// TIA Portal project "XSFW_TIA31001_B0_V15.1" (V15.1)

(* hardware
DEVICE "S7-1200 station_1"  S7-1200 Station
   slot 0: "Rack_0"  S7-1200 Rack  Rack  V1.0
   slot 1: "PLC_Divider"  CPU 1214C DC/DC/DC  6ES7 214-1AG40-0XB0  V4.2
   slot 2: "DI 16/DQ 16x24VDC_1"  6ES7 223-1BL32-0XB0  V2.0
   slot 3: "AI 4x13BIT/AQ 2x14BIT_1"  6ES7 234-4HE32-0XB0  V2.0
   slot 101: "CM 1242-5"  CM 1242-5  6GK7 242-5DX30-0XE0  V1.0
DEVICE "CSM"  SCALANCE X-Station
   slot 0: "Bastidor SCALANCE X"  Rail
   slot 0: "Switch"  6GK7 277-1AA00-0AA0
DEVICE "HMI_1"  KTP700 Basic PN
   slot 0: "HMI_1"  KTP700 Basic PN  6AV2 123-2GB03-0AX0  15.0.0.0
   slot 1: "HMI_RT_1"  KTP700 Basic PN  6AV2 123-2GB03-0AX0  15.0.0.0
   slot 5: "HMI_1.IE_CP_1"  PROFINET Interface  15.0.0.0
      slot 1: "Interfaz PROFINET_1"  PROFINET Interface
         slot 1: "Port_1"  Port
DEVICE "Dispositivo GSD_1"  GSD.Device.PN
   slot 0: "Rack"  Rack  V1.0
   slot 0: "V90-X"  SINAMICS V90 PN V1.0  6SL3 210-5Fxxx-xxFx  V1.00
      slot 0: "SINAMICS V90 PN V1.0"  SINAMICS V90 PN V1.0
      slot 1: "PN-IO"  PN-IO
         slot 1: "Puerto 1"  Port 1
         slot 2: "Puerto 2"  Port 2
      slot 1: "Drive"  Drive
         slot 0: "Punto de acceso a módulo"  Module Access Point
         slot 1: "sin PROFIsafe"  without PROFIsafe
   slot 2: "Telegrama estándar 3, PZD-5/9"  Standard telegram 3, PZD-5/9
DEVICE "Dispositivo GSD_2"  GSD.Device.PN
   slot 0: "Rack"  Rack  V1.0
   slot 0: "V90-Y"  SINAMICS V90 PN V1.0  6SL3 210-5Fxxx-xxFx  V1.00
      slot 0: "SINAMICS V90 PN V1.0"  SINAMICS V90 PN V1.0
      slot 1: "PN-IO"  PN-IO
         slot 1: "Puerto 1"  Port 1
         slot 2: "Puerto 2"  Port 2
      slot 1: "Drive"  Drive
         slot 0: "Punto de acceso a módulo"  Module Access Point
         slot 1: "sin PROFIsafe"  without PROFIsafe
   slot 2: "Telegrama estándar 3, PZD-5/9"  Standard telegram 3, PZD-5/9
*)

// ===== PLC "PLC_Divider"  CPU 1214C DC/DC/DC =====

VAR_GLOBAL   // PLC tag table "Tabla de variables estándar"
   "iCntBot" AT %I0.3 : Bool;
   "iSnsBotBaj" AT %I0.4 : Bool;
   "iSnsBotAlt" AT %I0.5 : Bool;
   "iCH_A" AT %I0.0 : Bool;
   "iCH_B" AT %I0.1 : Bool;
   "iCH_Z" AT %I0.2 : Bool;
   "iSns_Ch1Full" AT %I0.6 : Bool;
   "iSns_Ch2Full" AT %I3.6 : Bool;
   "iSns_Ch3Full" AT %I3.7 : Bool;
   "iSign_HabInv" AT %I3.0 : Bool;
   "iPul_Marcha" AT %I3.1 : Bool;
   "iPul_Parada" AT %I3.2 : Bool;
   "iPul_Rst" AT %I3.3 : Bool;
   "iProt_Abiertas" AT %I3.4 : Bool;
   "iTrip_Inverter" AT %I3.5 : Bool;
   "iRef_Analog" AT %IW54 : Int;
   "qRev_Alarma" AT %Q0.0 : Bool;
   "qSem_Verde" AT %Q0.1 : Bool;
   "qSem_rojo" AT %Q0.2 : Bool;
   "qTest_Marcha" AT %Q0.3 : Bool;
   "qRes_Alarma" AT %Q0.4 : Bool;
   "qRes_Inversor" AT %Q0.5 : Bool;
   "qFwd_Inversor" AT %Q0.6 : Bool;
   "qTrig_2" AT %Q0.7 : Bool;
   "qSign_Marcha" AT %Q1.0 : Bool;
   "qSign_Falla" AT %Q1.1 : Bool;
   "qTrig_1" AT %Q2.0 : Bool;
   "qTrig_22" AT %Q2.1 : Bool;
   "qRef_Analog" AT %IW82 : Int;
   "System_Byte" AT %MB1 : Byte;
   "FirstScan" AT %M1.0 : Bool;
   "DiagStatusUpdate" AT %M1.1 : Bool;
   "AlwaysTRUE" AT %M1.2 : Bool;
   "AlwaysFALSE" AT %M1.3 : Bool;
   "Clock_Byte" AT %MB0 : Byte;
   "Clock_10Hz" AT %M0.0 : Bool;
   "Clock_5Hz" AT %M0.1 : Bool;
   "Clock_2.5Hz" AT %M0.2 : Bool;
   "Clock_2Hz" AT %M0.3 : Bool;
   "Clock_1.25Hz" AT %M0.4 : Bool;
   "Clock_1Hz" AT %M0.5 : Bool;
   "Clock_0.625Hz" AT %M0.6 : Bool;
   "Clock_0.5Hz" AT %M0.7 : Bool;
   "Eje_Y_Drive_OUT" AT %Q74.0 : "PD_TEL3_OUT";
   "Eje_1_Drive_IN" AT %I68.0 : "PD_TEL3_IN";
   "Eje_1_Drive_OUT" AT %Q64.0 : "PD_TEL3_OUT";
   "MMovX" AT %M850.0 : Bool;
   "MMovXN" AT %M850.1 : Bool;
   "MMov2X" AT %M850.2 : Bool;
   "MMov2XN" AT %M850.3 : Bool;
   "MMovY" AT %M850.4 : Bool;
   "MMovYN" AT %M850.5 : Bool;
   "Eje_Y_Drive_IN(1)" AT %I86.0 : "PD_TEL3_IN";
   "Marca_Reset" AT %M103.0 : Bool;
   "SR_AlarmaOn" AT %M103.1 : Bool;
   "iHsc_Z" AT %ID1000 : DInt;
   "Hsc_Za" AT %MD20 : DInt;
   "Contando" AT %M150.0 : Bool;
   "Halt_Motor" AT %M150.2 : Bool;
   "Band_E24" AT %M150.3 : Bool;
   "Band_E22" AT %M150.4 : Bool;
   "Band_E23" AT %M150.5 : Bool;
   "Hsc_Zb" AT %MD28 : DInt;
   "Hsc_sub" AT %MD32 : DInt;
   "Hsc_sub1" AT %MD36 : DInt;
   "Enc_hab" AT %E104.0 : Bool;
   "Enc_stop" AT %I104.1 : Bool;
   "iEnc_Word1" AT %IW104 : Word;
   "iEnc_Word2" AT %IW106 : Word;
   "iEnc_Word3" AT %IW108 : Word;
   "iEnc_Word4" AT %IW110 : Word;
   "qEnc_Word5" AT %QW104 : Word;
   "qEnc_Word6" AT %QW106 : Word;
   "qEnc_Word7" AT %QW108 : Word;
   "qEnc_Word8" AT %QW110 : Word;
   "iSns_FinCarrX1" AT %I2.0 : Bool;
   "iSns_FinCarrX2" AT %I2.1 : Bool;
   "iSns_FinCarrY1" AT %I2.2 : Bool;
   "iSns_FinCarrY2" AT %I2.3 : Bool;
END_VAR

VAR_GLOBAL   // PLC tag table "Alarmas"
   "Alarmas_1" AT %MW100 : Word;
   "ProteccionAbierta" AT %M100.0 : Bool;
   "BotellaCaida" AT %M100.1 : Bool;
   "Fin_Carrera_X" AT %M100.4 : Bool;
   "Fin_Carrera_Y" AT %M100.5 : Bool;
   "Trip_Inverter" AT %M100.2 : Bool;
   "Error_Velocidad" AT %M100.3 : Bool;
END_VAR

VAR_GLOBAL   // PLC tag table "Inicializaciòn"
   "Marcas para la inicializaciòn" AT %MW102 : Word;
   "Start" AT %M102.0 : Bool;
END_VAR

DATA_BLOCK "01_LINEA_Entradas-DB"   // DB1
{ S7_Optimized_Access := 'TRUE' }
VERSION : 0.1
   VAR
      Contador : Bool;   // Pulsador de marcha
      Sensor_Bajo : Bool;   // Pulsador de parada
      Sensor_Alto : Bool;   // Pulsador de marcha columna 4
      CH_A : Bool;   // Pulsador de parada de emergancia columna 4
      CH_B : Bool;   // Pulsador de marcha columna 6
      CH_Z : Bool;   // Pulsador de parada de emergancia columna 6
      Canal1_Full : Bool;   // Pulsador de marcha columna 9
      Canal2_Full : Bool;   // Pulsador de parada de emergancia columna 9
      Canal3_Full : Bool;   // Pulsador de marcha columna 11
      Hab_Inverter : Bool;   // Pulsador de parada de emergancia columna 11
      Marcha : Bool;   // Pulsador de marcha columna 12
      Parada : Bool;   // Pulsador de parada de emergancia columna 12
      Reset : Bool;   // Pulsador de parada de emergancia del tablero general
      Protecciones_Abiertas : Bool;   // Pulsador de parada de emergencia del tablero de la fosa
      Trip_Inverter : Bool;   // Señal de falla del variador
      Enc_andando : Bool;
      Enc_parada : Bool;
   END_VAR
BEGIN
END_DATA_BLOCK

DATA_BLOCK "02_LINEA_Salidas-DB"   // DB2
{ S7_Optimized_Access := 'TRUE' }
VERSION : 0.1
   VAR
      Alarma_Sonora : Bool;   // Marcha para el variador
      Semaforo_Verde : Bool;   // Sentido adelante variador
      Semaforo_Rojo : Bool;   // Sentido atras variador
      Testigo_Marcha : Bool;   // Indicador sonoro
      Reset_Alarma : Bool;   // Indicador de linea en marcha
      Reset_Inverter : Bool;   // Indicador de linea parada
      Avance_Inverter : Bool;   // Buzzer de la baliza del tablero principal
      Trigger_2 : Bool;   // Lampara verde de la baliza del tablero principal
      EnMarcha : Bool;   // Lampara roja de la baliza del tablero principal
      EnFalla : Bool;   // Lampara amarilla de la baliza del tablero principal
      Trigger_11 : Bool;
      Trigger_22 : Bool;
      Ref_20mA : Int;
   END_VAR
BEGIN
END_DATA_BLOCK

DATA_BLOCK "MotorInverter"   // DB5
{ S7_Optimized_Access := 'TRUE' }
VERSION : 0.1
// stored: InstanceOfName Motor Simple
"Motor Simple"
BEGIN
END_DATA_BLOCK

DATA_BLOCK "FB_INC_GENERAL_DB"   // DB7
{ S7_Optimized_Access := 'FALSE' }
VERSION : 0.1
// stored: InstanceOfName FB_INC_GENERAL
"FB_INC_GENERAL"
BEGIN
END_DATA_BLOCK

DATA_BLOCK "Cuentas_Matematicas1_DB"   // DB15
{ S7_Optimized_Access := 'TRUE' }
VERSION : 0.1
   VAR
      MovXNeg : Real := 0.0;
      Mov2X : Real := 0.0;
      Mov2XNeg : Real := 0.0;
      MovYNeg : Real := 0.0;
   END_VAR
BEGIN
END_DATA_BLOCK

DATA_BLOCK "FB_GENERAL_DB"   // DB17
{ S7_Optimized_Access := 'FALSE' }
VERSION : 0.1
// stored: InstanceOfName FB_SUB_1_GENERAL
"FB_SUB_1_GENERAL"
BEGIN
END_DATA_BLOCK

DATA_BLOCK "Cuentas_Matematicas1_DB_1"   // DB20
{ S7_Optimized_Access := 'TRUE' }
VERSION : 0.1
// stored: InstanceOfName Cuentas_Matematicas1
"Cuentas_Matematicas1"
BEGIN
END_DATA_BLOCK

DATA_BLOCK "DB_Encajonadora"   // DB28
{ S7_Optimized_Access := 'TRUE' }
VERSION : 0.1
   VAR
      Word1 : Word;   // bit 0 y 1 para guardar estado de encajonadora
      Word2 : Word;
      Word3 : Word;
      Word4 : Word;
      Word5 : Word;
      Word6 : Word;
      Word7 : Word;
      Word8 : Word;
   END_VAR
BEGIN
END_DATA_BLOCK

DATA_BLOCK "FB_SUB_1_GENERAL_DB"   // DB35
{ S7_Optimized_Access := 'FALSE' }
VERSION : 0.1
// stored: InstanceOfName FB_SUB_1_GENERAL
"FB_SUB_1_GENERAL"
BEGIN
END_DATA_BLOCK

DATA_BLOCK "FB_SUB_0_GENERAL_DB"   // DB36
{ S7_Optimized_Access := 'TRUE' }
VERSION : 0.1
// stored: InstanceOfName FB_SUB_0_GENERAL
"FB_SUB_0_GENERAL"
BEGIN
END_DATA_BLOCK

DATA_BLOCK "DB_SUB_1_GENERAL"   // DB100
{ S7_Optimized_Access := 'FALSE' }
VERSION : 0.1
// stored: InstanceOfName FB_SUB_1_GENERAL
"FB_SUB_1_GENERAL"
BEGIN
END_DATA_BLOCK

// folder: COMANDOS

DATA_BLOCK "DB_SUB_0_COM_GENERAL"   // DB600
{ S7_Optimized_Access := 'FALSE' }
VERSION : 0.1
   VAR
      ManipEsperaCarro : Bool;
      RecepCarroConfir : Bool;
      SalidaEsperaCarro1 : Bool;
      SalidaEsperaCarro2 : Bool;
      TengoCarroEnPortacarro : Bool;
      ReconocimientoAlarmas : Bool;
   END_VAR
BEGIN
END_DATA_BLOCK

// folder: INCIDENTES

DATA_BLOCK "DB_INC_GENERAL"   // DB500
{ S7_Optimized_Access := 'FALSE' }
VERSION : 0.1
// stored: InstanceOfName FB_INC_GENERAL
"FB_INC_GENERAL"
BEGIN
END_DATA_BLOCK

// folder: PUESTA EN MARCHA

DATA_BLOCK "DB_PUESTA_MARCHA"   // DB10
{ S7_Optimized_Access := 'TRUE' }
VERSION : 0.1
   VAR RETAIN
      MovYmm : Real := 30.0;
      MovXmm : Real := 30.0;
   END_VAR
   VAR
      TChFull : Time := T#1S;
   END_VAR
BEGIN
END_DATA_BLOCK

// folder: System blocks/Program resources

DATA_BLOCK "IEC_Counter_0_DB"   // DB6
{ S7_Optimized_Access := 'TRUE' }
AUTHOR : Simatic
FAMILY : IEC
NAME : CNTR
VERSION : 1.0
// stored: InstanceOfName IEC_COUNTER
"IEC_COUNTER"
BEGIN
END_DATA_BLOCK

DATA_BLOCK "IEC_Counter_1_DB"   // DB8
{ S7_Optimized_Access := 'TRUE' }
AUTHOR : Simatic
FAMILY : IEC
NAME : CNTR
VERSION : 1.0
// stored: InstanceOfName IEC_COUNTER
"IEC_COUNTER"
BEGIN
END_DATA_BLOCK

DATA_BLOCK "IEC_Counter_2_DB"   // DB9
{ S7_Optimized_Access := 'TRUE' }
AUTHOR : Simatic
FAMILY : IEC
NAME : CNTR
VERSION : 1.0
// stored: InstanceOfName IEC_COUNTER
"IEC_COUNTER"
BEGIN
END_DATA_BLOCK

DATA_BLOCK "IEC_Timer_ChFull"   // DB11
{ S7_Optimized_Access := 'TRUE' }
AUTHOR : Simatic
FAMILY : IEC
NAME : IEC_TMR
VERSION : 1.0
// stored: InstanceOfName IEC_TIMER
"IEC_TIMER"
BEGIN
END_DATA_BLOCK

DATA_BLOCK "IEC_Timer_0_DB_1"   // DB30
{ S7_Optimized_Access := 'TRUE' }
AUTHOR : Simatic
FAMILY : IEC
NAME : IEC_TMR
VERSION : 1.0
// stored: InstanceOfName IEC_TIMER
"IEC_TIMER"
BEGIN
END_DATA_BLOCK

DATA_BLOCK "IEC_Timer_0_DB_2"   // DB31
{ S7_Optimized_Access := 'TRUE' }
AUTHOR : Simatic
FAMILY : IEC
NAME : IEC_TMR
VERSION : 1.0
// stored: InstanceOfName IEC_TIMER
"IEC_TIMER"
BEGIN
END_DATA_BLOCK

DATA_BLOCK "IEC_Timer_0_DB_3"   // DB32
{ S7_Optimized_Access := 'TRUE' }
AUTHOR : Simatic
FAMILY : IEC
NAME : IEC_TMR
VERSION : 1.0
// stored: InstanceOfName IEC_TIMER
"IEC_TIMER"
BEGIN
END_DATA_BLOCK

DATA_BLOCK "IEC_Timer_0_DB_4"   // DB33
{ S7_Optimized_Access := 'TRUE' }
AUTHOR : Simatic
FAMILY : IEC
NAME : IEC_TMR
VERSION : 1.0
// stored: InstanceOfName IEC_TIMER
"IEC_TIMER"
BEGIN
END_DATA_BLOCK

DATA_BLOCK "IEC_Timer_0_DB_5"   // DB34
{ S7_Optimized_Access := 'TRUE' }
AUTHOR : Simatic
FAMILY : IEC
NAME : IEC_TMR
VERSION : 1.0
// stored: InstanceOfName IEC_TIMER
"IEC_TIMER"
BEGIN
END_DATA_BLOCK

// folder: VISUALIZACION

DATA_BLOCK "DB_VIS_GENERAL"   // DB800
{ S7_Optimized_Access := 'FALSE' }
VERSION : 0.1
   VAR
      CantBot : Int;
      AlarmaProtecciòn : Bool;
      AlarmaBotellaCaida : Bool;
      MC_Pwr_EnX : Bool;
      MC_Pwrt_EnY : Bool;
      MC_Res_ExX : Bool;
      MC_Res_ExY : Bool;
      MC_JogFwd_X : Bool;
      MC_JogFwd_Y : Bool;
      MC_JogBwd_X : Bool;
      MC_JogBwd_Y : Bool;
      HomingOk : Bool;
      Reset : Bool;
      Start : Bool;
   END_VAR
BEGIN
END_DATA_BLOCK

// folder: (top level)

DATA_BLOCK "Eje_Y"   // DB4, Motion_DB
{ S7_Optimized_Access := 'TRUE' }
AUTHOR : SIMATIC
FAMILY : BasicMC
NAME : TO_PosAx
VERSION : 6.0
// stored: InstanceOfName TO_PositioningAxis
"TO_PositioningAxis"
BEGIN
   // Axis.Encoder.TelegramAddressOutCU = %Q74.0
   // Axis.Encoder.TelegramAddressInCU = %I86.0
   // Axis.Encoder.DoNameCU = V90-Y.Drive_Encóder1
   // Axis.Drive.TelegramAddressOutCU = %Q74.0
   // Axis.Drive.TelegramAddressInCU = %I86.0
   // Axis.Drive.TelegramType = 2
   // Axis.Drive.DoNameCU = V90-Y.Drive
   // Axis.LengthUnitNormalized.Time = 1
   // Axis.LengthUnitNormalized.Distance = -2
   // Axis.Encoder.SelectedHscIndexCU = -1
   // Axis.Encoder.DbTypeCU = Classic
   // Axis.Drive.DbTypeCU = Classic
END_DATA_BLOCK

DATA_BLOCK "Eje_X"   // DB12, Motion_DB
{ S7_Optimized_Access := 'TRUE' }
AUTHOR : SIMATIC
FAMILY : BasicMC
NAME : TO_PosAx
VERSION : 6.0
// stored: InstanceOfName TO_PositioningAxis
"TO_PositioningAxis"
BEGIN
   // Axis.Encoder.TelegramAddressOutCU = %Q64.0
   // Axis.Encoder.TelegramAddressInCU = %I68.0
   // Axis.Encoder.DoNameCU = V90-X.Drive_Encóder1
   // Axis.Drive.TelegramAddressOutCU = %Q64.0
   // Axis.Drive.TelegramAddressInCU = %I68.0
   // Axis.Drive.TelegramType = 2
   // Axis.Drive.DoNameCU = V90-X.Drive
   // Axis.LengthUnitNormalized.Distance = 1013
   // Axis.Encoder.SelectedHscIndexCU = -1
   // Axis.Encoder.DbTypeCU = Classic
   // Axis.Drive.DbTypeCU = Classic
END_DATA_BLOCK

FUNCTION_BLOCK "Cuentas_Matematicas1"   // FB1, LAD
TITLE = ---------------------------Calculo de distancias----------------------------------------
{ S7_Optimized_Access := 'TRUE' }
VERSION : 0.1
BEGIN

REGION Network 1: Movimiento negativo en X
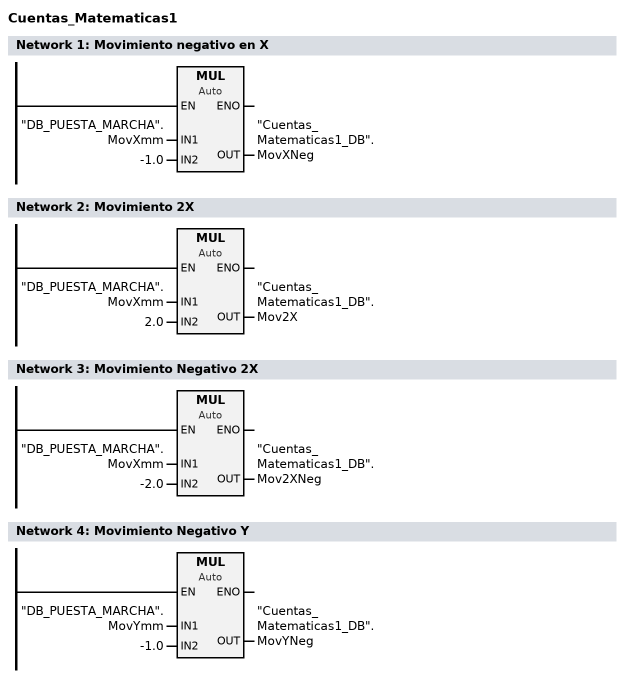
   RUNG wire#powerrail
      Mul(in1 := "DB_PUESTA_MARCHA".MovXmm, in2 := -1.0, out => "Cuentas_Matematicas1_DB".MovXNeg)
   END_RUNG
   // the same network as SCL:
   "Cuentas_Matematicas1_DB".MovXNeg := "DB_PUESTA_MARCHA".MovXmm * (-1.0);
END_REGION

REGION Network 2: Movimiento 2X
   RUNG wire#powerrail
      Mul(in1 := "DB_PUESTA_MARCHA".MovXmm, in2 := 2.0, out => "Cuentas_Matematicas1_DB".Mov2X)
   END_RUNG
   // the same network as SCL:
   "Cuentas_Matematicas1_DB".Mov2X := "DB_PUESTA_MARCHA".MovXmm * 2.0;
END_REGION

REGION Network 3: Movimiento Negativo 2X
   RUNG wire#powerrail
      Mul(in1 := "DB_PUESTA_MARCHA".MovXmm, in2 := -2.0, out => "Cuentas_Matematicas1_DB".Mov2XNeg)
   END_RUNG
   // the same network as SCL:
   "Cuentas_Matematicas1_DB".Mov2XNeg := "DB_PUESTA_MARCHA".MovXmm * (-2.0);
END_REGION

REGION Network 4: Movimiento Negativo Y
   RUNG wire#powerrail
      Mul(in1 := "DB_PUESTA_MARCHA".MovYmm, in2 := -1.0, out => "Cuentas_Matematicas1_DB".MovYNeg)
   END_RUNG
   // the same network as SCL:
   "Cuentas_Matematicas1_DB".MovYNeg := "DB_PUESTA_MARCHA".MovYmm * (-1.0);
END_REGION
END_FUNCTION_BLOCK

FUNCTION_BLOCK "FB_SUB_0_GENERAL"   // FB3, LAD
{ S7_Optimized_Access := 'TRUE' }
VERSION : 0.1
BEGIN

REGION Network 1
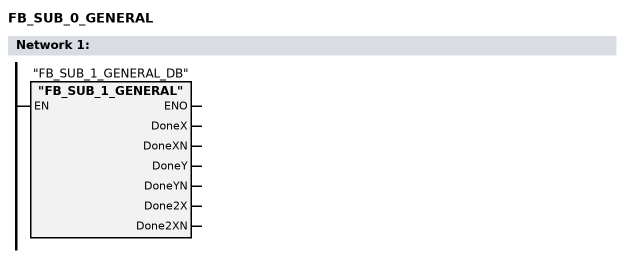
   RUNG wire#powerrail
      "FB_SUB_1_GENERAL_DB"(DoneX =>, DoneXN =>, DoneY =>, DoneYN =>, Done2X =>, Done2XN =>)
   END_RUNG
   // the same network as SCL:
   "FB_SUB_1_GENERAL_DB"();   // "FB_SUB_1_GENERAL"
END_REGION
END_FUNCTION_BLOCK

FUNCTION_BLOCK "FB_SUB_1_GENERAL"   // FB100, LAD
{ S7_Optimized_Access := 'FALSE' }
VERSION : 0.1
   VAR_OUTPUT
      DoneX : Bool;
      DoneXN : Bool;
      DoneY : Bool;
      DoneYN : Bool;
      Done2X : Bool;
      Done2XN : Bool;
   END_VAR
   VAR
      Estados : Array[0..32] of Bool;
      Concatenadoras : Array[0..32] of Bool;
      Prioritarias : Array[0..32] of Bool;
      Error_Concatenadoras : Bool;
      Error_Prioritarias : Bool;
      Cuenta_1 : Bool;
      Cuenta_2 : Bool;
      Cuenta_3 : Bool;
      "Cont_Botellas/2" : Int;
   END_VAR
BEGIN

REGION Network 1: Inicializaciòn
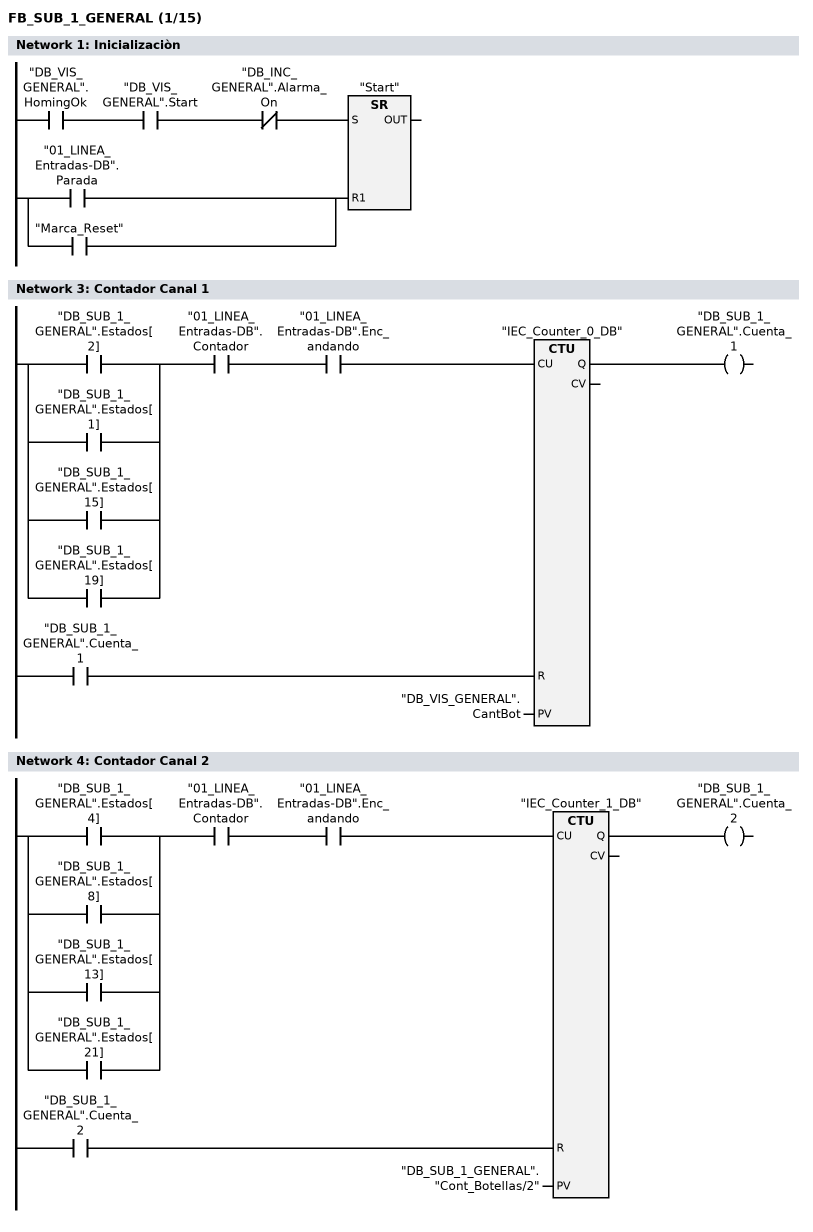
   RUNG wire#powerrail
      Contact( "DB_VIS_GENERAL".HomingOk )
      Contact( "DB_VIS_GENERAL".Start )
      I_Contact( "DB_INC_GENERAL".Alarma_On )
      S_SR(operand := "Start", r1 := wire#w1)
   END_RUNG
   RUNG wire#powerrail
      Contact( "01_LINEA_Entradas-DB".Parada )
   END_RUNG wire#w1
   RUNG wire#powerrail
      Contact( "Marca_Reset" )
   END_RUNG wire#w1
   // the same network as SCL:
   IF "DB_VIS_GENERAL".HomingOk AND "DB_VIS_GENERAL".Start AND NOT "DB_INC_GENERAL".Alarma_On THEN
       "Start" := TRUE;   // SR flip-flop
   END_IF;
   IF "01_LINEA_Entradas-DB".Parada OR "Marca_Reset" THEN "Start" := FALSE; END_IF;
END_REGION

REGION Network 2: -----------------OTROS---------------
END_REGION

REGION Network 3: Contador Canal 1
   "IEC_Counter_0_DB".CTU(CU := ("DB_SUB_1_GENERAL".Estados[2] OR "DB_SUB_1_GENERAL".Estados[1] OR "DB_SUB_1_GENERAL".Estados[15] OR "DB_SUB_1_GENERAL".Estados[19]) AND "01_LINEA_Entradas-DB".Contador AND "01_LINEA_Entradas-DB".Enc_andando,
                          R := "DB_SUB_1_GENERAL".Cuenta_1,
                          PV := "DB_VIS_GENERAL".CantBot);
   "DB_SUB_1_GENERAL".Cuenta_1 := "IEC_Counter_0_DB".Q;
END_REGION

REGION Network 4: Contador Canal 2
   "IEC_Counter_1_DB".CTU(CU := ("DB_SUB_1_GENERAL".Estados[4] OR "DB_SUB_1_GENERAL".Estados[8] OR "DB_SUB_1_GENERAL".Estados[13] OR "DB_SUB_1_GENERAL".Estados[21]) AND "01_LINEA_Entradas-DB".Contador AND "01_LINEA_Entradas-DB".Enc_andando,
                          R := "DB_SUB_1_GENERAL".Cuenta_2,
                          PV := "DB_SUB_1_GENERAL"."Cont_Botellas/2");
   "DB_SUB_1_GENERAL".Cuenta_2 := "IEC_Counter_1_DB".Q;
END_REGION

REGION Network 5: CASO I CANAL 2
   // Caso en el cual CH1/2 no estan llenos y hay que repartir solo la mitad de las botellas en canal central
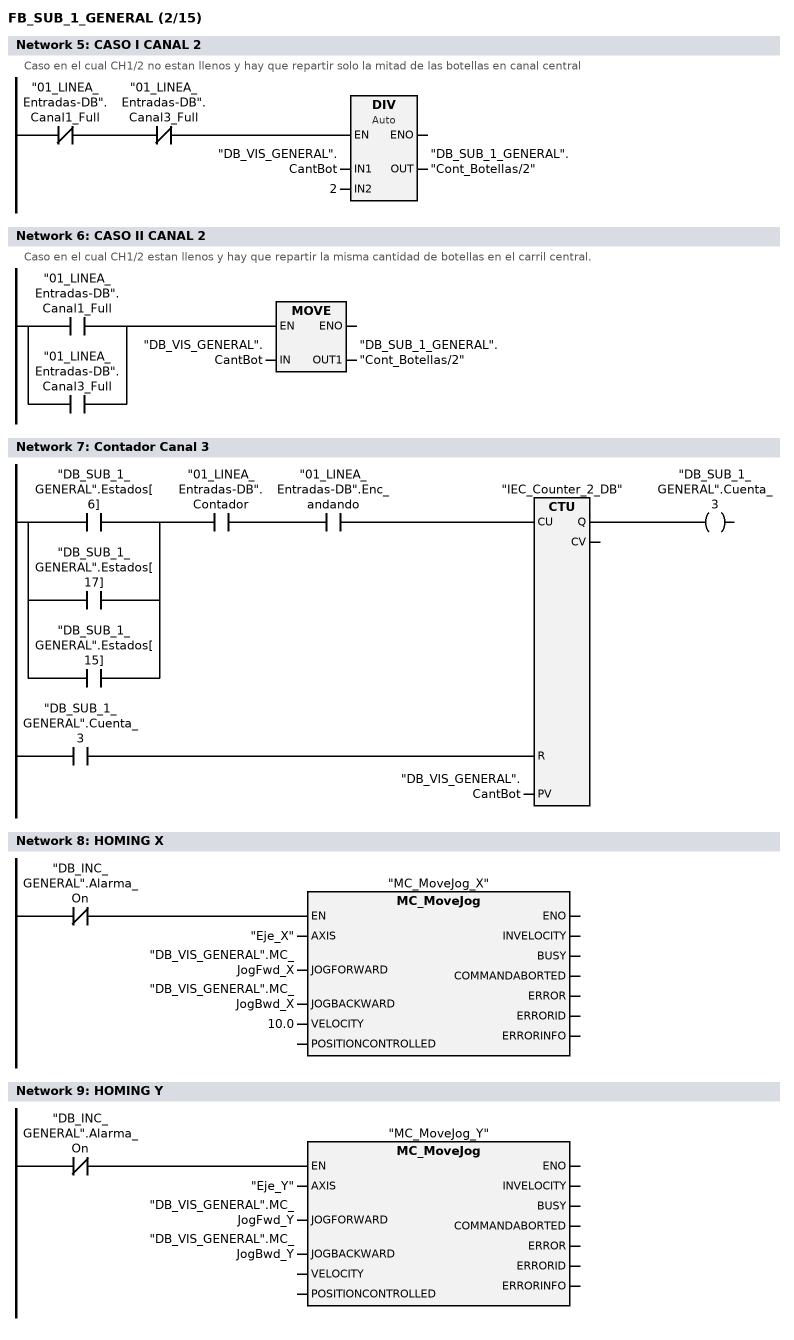
   RUNG wire#powerrail
      I_Contact( "01_LINEA_Entradas-DB".Canal1_Full )
      I_Contact( "01_LINEA_Entradas-DB".Canal3_Full )
      Div(in1 := "DB_VIS_GENERAL".CantBot, in2 := 2, out => "DB_SUB_1_GENERAL"."Cont_Botellas/2")
   END_RUNG
   // the same network as SCL:
   IF NOT "01_LINEA_Entradas-DB".Canal1_Full AND NOT "01_LINEA_Entradas-DB".Canal3_Full THEN
       "DB_SUB_1_GENERAL"."Cont_Botellas/2" := "DB_VIS_GENERAL".CantBot / 2;
   END_IF;
END_REGION

REGION Network 6: CASO II CANAL 2
   // Caso en el cual CH1/2 estan llenos y hay que repartir la misma cantidad de botellas en el carril central.
   RUNG wire#powerrail
      Contact( "01_LINEA_Entradas-DB".Canal1_Full )
      wire#w1
      Move(in := "DB_VIS_GENERAL".CantBot, out1 => "DB_SUB_1_GENERAL"."Cont_Botellas/2")
   END_RUNG
   RUNG wire#powerrail
      Contact( "01_LINEA_Entradas-DB".Canal3_Full )
   END_RUNG wire#w1
   // the same network as SCL:
   IF "01_LINEA_Entradas-DB".Canal1_Full OR "01_LINEA_Entradas-DB".Canal3_Full THEN
       "DB_SUB_1_GENERAL"."Cont_Botellas/2" := "DB_VIS_GENERAL".CantBot;
   END_IF;
END_REGION

REGION Network 7: Contador Canal 3
   "IEC_Counter_2_DB".CTU(CU := ("DB_SUB_1_GENERAL".Estados[6] OR "DB_SUB_1_GENERAL".Estados[17] OR "DB_SUB_1_GENERAL".Estados[15]) AND "01_LINEA_Entradas-DB".Contador AND "01_LINEA_Entradas-DB".Enc_andando,
                          R := "DB_SUB_1_GENERAL".Cuenta_3,
                          PV := "DB_VIS_GENERAL".CantBot);
   "DB_SUB_1_GENERAL".Cuenta_3 := "IEC_Counter_2_DB".Q;
END_REGION

REGION Network 8: HOMING X
   IF NOT "DB_INC_GENERAL".Alarma_On THEN
       "MC_MoveJog_X"(Axis := "Eje_X",   // MC_MoveJog
                      JogForward := "DB_VIS_GENERAL".MC_JogFwd_X,
                      JogBackward := "DB_VIS_GENERAL".MC_JogBwd_X,
                      Velocity := 10.0);
   END_IF;
END_REGION

REGION Network 9: HOMING Y
   IF NOT "DB_INC_GENERAL".Alarma_On THEN
       "MC_MoveJog_Y"(Axis := "Eje_Y",   // MC_MoveJog
                      JogForward := "DB_VIS_GENERAL".MC_JogFwd_Y,
                      JogBackward := "DB_VIS_GENERAL".MC_JogBwd_Y);
   END_IF;
END_REGION

REGION Network 10: --------------------Maquina de estados - 3 carriles-----------------
END_REGION

REGION Network 11: Concatenadora 1
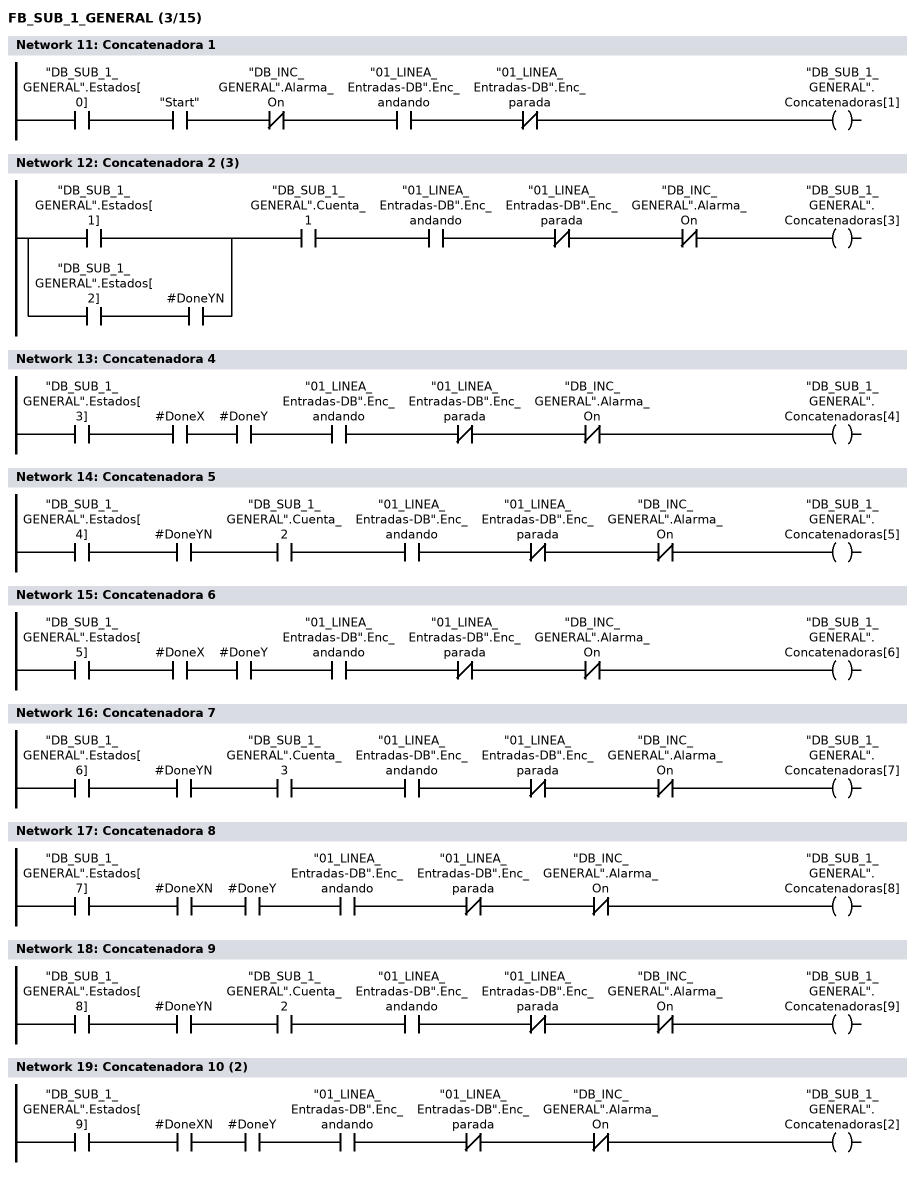
   RUNG wire#powerrail
      Contact( "DB_SUB_1_GENERAL".Estados[0] )
      Contact( "Start" )
      I_Contact( "DB_INC_GENERAL".Alarma_On )
      Contact( "01_LINEA_Entradas-DB".Enc_andando )
      I_Contact( "01_LINEA_Entradas-DB".Enc_parada )
      Coil( "DB_SUB_1_GENERAL".Concatenadoras[1] )
   END_RUNG
   // the same network as SCL:
   "DB_SUB_1_GENERAL".Concatenadoras[1] := "DB_SUB_1_GENERAL".Estados[0] AND "Start" AND NOT "DB_INC_GENERAL".Alarma_On AND "01_LINEA_Entradas-DB".Enc_andando AND NOT "01_LINEA_Entradas-DB".Enc_parada;
END_REGION

REGION Network 12: Concatenadora 2 (3)
   RUNG wire#powerrail
      Contact( "DB_SUB_1_GENERAL".Estados[1] )
      wire#w1
      Contact( "DB_SUB_1_GENERAL".Cuenta_1 )
      Contact( "01_LINEA_Entradas-DB".Enc_andando )
      I_Contact( "01_LINEA_Entradas-DB".Enc_parada )
      I_Contact( "DB_INC_GENERAL".Alarma_On )
      Coil( "DB_SUB_1_GENERAL".Concatenadoras[3] )
   END_RUNG
   RUNG wire#powerrail
      Contact( "DB_SUB_1_GENERAL".Estados[2] )
      Contact( #DoneYN )
   END_RUNG wire#w1
   // the same network as SCL:
   "DB_SUB_1_GENERAL".Concatenadoras[3] := ("DB_SUB_1_GENERAL".Estados[1] OR ("DB_SUB_1_GENERAL".Estados[2] AND #DoneYN)) AND "DB_SUB_1_GENERAL".Cuenta_1 AND "01_LINEA_Entradas-DB".Enc_andando AND NOT "01_LINEA_Entradas-DB".Enc_parada AND NOT "DB_INC_GENERAL".Alarma_On;
END_REGION

REGION Network 13: Concatenadora 4
   RUNG wire#powerrail
      Contact( "DB_SUB_1_GENERAL".Estados[3] )
      Contact( #DoneX )
      Contact( #DoneY )
      Contact( "01_LINEA_Entradas-DB".Enc_andando )
      I_Contact( "01_LINEA_Entradas-DB".Enc_parada )
      I_Contact( "DB_INC_GENERAL".Alarma_On )
      Coil( "DB_SUB_1_GENERAL".Concatenadoras[4] )
   END_RUNG
   // the same network as SCL:
   "DB_SUB_1_GENERAL".Concatenadoras[4] := "DB_SUB_1_GENERAL".Estados[3] AND #DoneX AND #DoneY AND "01_LINEA_Entradas-DB".Enc_andando AND NOT "01_LINEA_Entradas-DB".Enc_parada AND NOT "DB_INC_GENERAL".Alarma_On;
END_REGION

REGION Network 14: Concatenadora 5
   RUNG wire#powerrail
      Contact( "DB_SUB_1_GENERAL".Estados[4] )
      Contact( #DoneYN )
      Contact( "DB_SUB_1_GENERAL".Cuenta_2 )
      Contact( "01_LINEA_Entradas-DB".Enc_andando )
      I_Contact( "01_LINEA_Entradas-DB".Enc_parada )
      I_Contact( "DB_INC_GENERAL".Alarma_On )
      Coil( "DB_SUB_1_GENERAL".Concatenadoras[5] )
   END_RUNG
   // the same network as SCL:
   "DB_SUB_1_GENERAL".Concatenadoras[5] := "DB_SUB_1_GENERAL".Estados[4] AND #DoneYN AND "DB_SUB_1_GENERAL".Cuenta_2 AND "01_LINEA_Entradas-DB".Enc_andando AND NOT "01_LINEA_Entradas-DB".Enc_parada AND NOT "DB_INC_GENERAL".Alarma_On;
END_REGION

REGION Network 15: Concatenadora 6
   RUNG wire#powerrail
      Contact( "DB_SUB_1_GENERAL".Estados[5] )
      Contact( #DoneX )
      Contact( #DoneY )
      Contact( "01_LINEA_Entradas-DB".Enc_andando )
      I_Contact( "01_LINEA_Entradas-DB".Enc_parada )
      I_Contact( "DB_INC_GENERAL".Alarma_On )
      Coil( "DB_SUB_1_GENERAL".Concatenadoras[6] )
   END_RUNG
   // the same network as SCL:
   "DB_SUB_1_GENERAL".Concatenadoras[6] := "DB_SUB_1_GENERAL".Estados[5] AND #DoneX AND #DoneY AND "01_LINEA_Entradas-DB".Enc_andando AND NOT "01_LINEA_Entradas-DB".Enc_parada AND NOT "DB_INC_GENERAL".Alarma_On;
END_REGION

REGION Network 16: Concatenadora 7
   RUNG wire#powerrail
      Contact( "DB_SUB_1_GENERAL".Estados[6] )
      Contact( #DoneYN )
      Contact( "DB_SUB_1_GENERAL".Cuenta_3 )
      Contact( "01_LINEA_Entradas-DB".Enc_andando )
      I_Contact( "01_LINEA_Entradas-DB".Enc_parada )
      I_Contact( "DB_INC_GENERAL".Alarma_On )
      Coil( "DB_SUB_1_GENERAL".Concatenadoras[7] )
   END_RUNG
   // the same network as SCL:
   "DB_SUB_1_GENERAL".Concatenadoras[7] := "DB_SUB_1_GENERAL".Estados[6] AND #DoneYN AND "DB_SUB_1_GENERAL".Cuenta_3 AND "01_LINEA_Entradas-DB".Enc_andando AND NOT "01_LINEA_Entradas-DB".Enc_parada AND NOT "DB_INC_GENERAL".Alarma_On;
END_REGION

REGION Network 17: Concatenadora 8
   RUNG wire#powerrail
      Contact( "DB_SUB_1_GENERAL".Estados[7] )
      Contact( #DoneXN )
      Contact( #DoneY )
      Contact( "01_LINEA_Entradas-DB".Enc_andando )
      I_Contact( "01_LINEA_Entradas-DB".Enc_parada )
      I_Contact( "DB_INC_GENERAL".Alarma_On )
      Coil( "DB_SUB_1_GENERAL".Concatenadoras[8] )
   END_RUNG
   // the same network as SCL:
   "DB_SUB_1_GENERAL".Concatenadoras[8] := "DB_SUB_1_GENERAL".Estados[7] AND #DoneXN AND #DoneY AND "01_LINEA_Entradas-DB".Enc_andando AND NOT "01_LINEA_Entradas-DB".Enc_parada AND NOT "DB_INC_GENERAL".Alarma_On;
END_REGION

REGION Network 18: Concatenadora 9
   RUNG wire#powerrail
      Contact( "DB_SUB_1_GENERAL".Estados[8] )
      Contact( #DoneYN )
      Contact( "DB_SUB_1_GENERAL".Cuenta_2 )
      Contact( "01_LINEA_Entradas-DB".Enc_andando )
      I_Contact( "01_LINEA_Entradas-DB".Enc_parada )
      I_Contact( "DB_INC_GENERAL".Alarma_On )
      Coil( "DB_SUB_1_GENERAL".Concatenadoras[9] )
   END_RUNG
   // the same network as SCL:
   "DB_SUB_1_GENERAL".Concatenadoras[9] := "DB_SUB_1_GENERAL".Estados[8] AND #DoneYN AND "DB_SUB_1_GENERAL".Cuenta_2 AND "01_LINEA_Entradas-DB".Enc_andando AND NOT "01_LINEA_Entradas-DB".Enc_parada AND NOT "DB_INC_GENERAL".Alarma_On;
END_REGION

REGION Network 19: Concatenadora 10 (2)
   RUNG wire#powerrail
      Contact( "DB_SUB_1_GENERAL".Estados[9] )
      Contact( #DoneXN )
      Contact( #DoneY )
      Contact( "01_LINEA_Entradas-DB".Enc_andando )
      I_Contact( "01_LINEA_Entradas-DB".Enc_parada )
      I_Contact( "DB_INC_GENERAL".Alarma_On )
      Coil( "DB_SUB_1_GENERAL".Concatenadoras[2] )
   END_RUNG
   // the same network as SCL:
   "DB_SUB_1_GENERAL".Concatenadoras[2] := "DB_SUB_1_GENERAL".Estados[9] AND #DoneXN AND #DoneY AND "01_LINEA_Entradas-DB".Enc_andando AND NOT "01_LINEA_Entradas-DB".Enc_parada AND NOT "DB_INC_GENERAL".Alarma_On;
END_REGION

REGION Network 20: ---------------Maquina de estado - 2 carriles -------------
END_REGION

REGION Network 21: Concatenadora 11
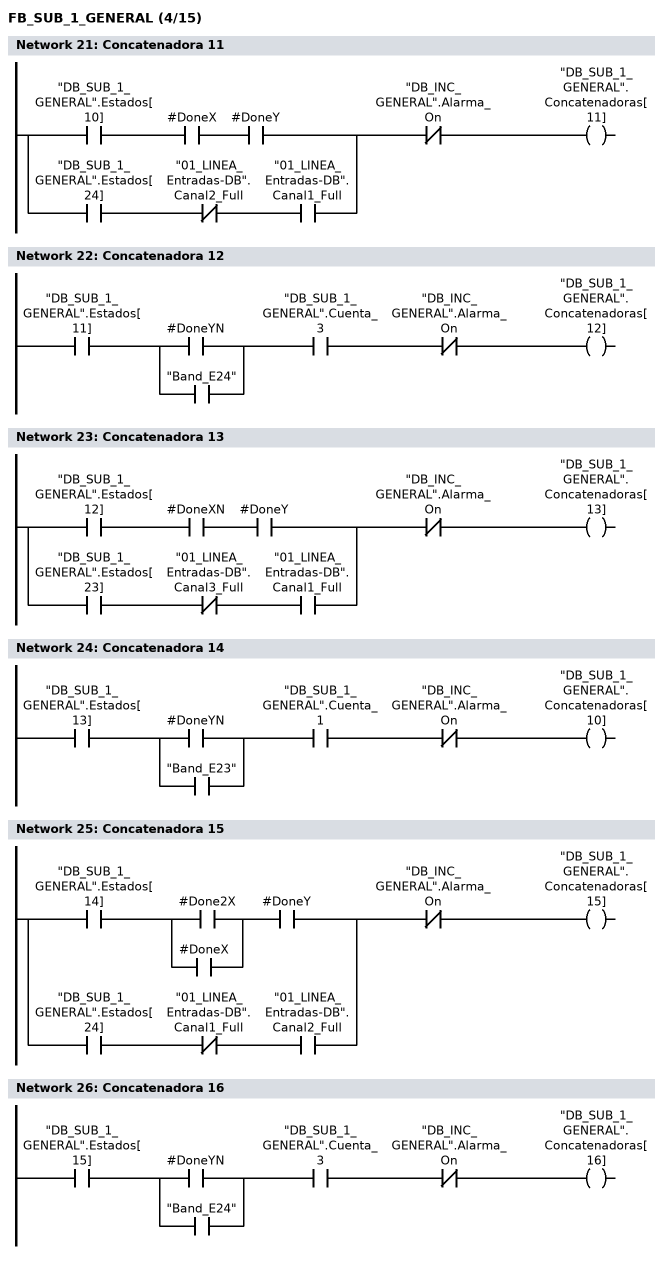
   RUNG wire#powerrail
      Contact( "DB_SUB_1_GENERAL".Estados[10] )
      Contact( #DoneX )
      Contact( #DoneY )
      wire#w1
      I_Contact( "DB_INC_GENERAL".Alarma_On )
      Coil( "DB_SUB_1_GENERAL".Concatenadoras[11] )
   END_RUNG
   RUNG wire#powerrail
      Contact( "DB_SUB_1_GENERAL".Estados[24] )
      I_Contact( "01_LINEA_Entradas-DB".Canal2_Full )
      Contact( "01_LINEA_Entradas-DB".Canal1_Full )
   END_RUNG wire#w1
   // the same network as SCL:
   "DB_SUB_1_GENERAL".Concatenadoras[11] := (("DB_SUB_1_GENERAL".Estados[10] AND #DoneX AND #DoneY) OR ("DB_SUB_1_GENERAL".Estados[24] AND NOT "01_LINEA_Entradas-DB".Canal2_Full AND "01_LINEA_Entradas-DB".Canal1_Full)) AND NOT "DB_INC_GENERAL".Alarma_On;
END_REGION

REGION Network 22: Concatenadora 12
   RUNG wire#powerrail
      Contact( "DB_SUB_1_GENERAL".Estados[11] )
      wire#w1
      Contact( #DoneYN )
      wire#w2
      Contact( "DB_SUB_1_GENERAL".Cuenta_3 )
      I_Contact( "DB_INC_GENERAL".Alarma_On )
      Coil( "DB_SUB_1_GENERAL".Concatenadoras[12] )
   END_RUNG
   RUNG wire#w1
      Contact( "Band_E24" )
   END_RUNG wire#w2
   // the same network as SCL:
   "DB_SUB_1_GENERAL".Concatenadoras[12] := "DB_SUB_1_GENERAL".Estados[11] AND (#DoneYN OR "Band_E24") AND "DB_SUB_1_GENERAL".Cuenta_3 AND NOT "DB_INC_GENERAL".Alarma_On;
END_REGION

REGION Network 23: Concatenadora 13
   RUNG wire#powerrail
      Contact( "DB_SUB_1_GENERAL".Estados[12] )
      Contact( #DoneXN )
      Contact( #DoneY )
      wire#w1
      I_Contact( "DB_INC_GENERAL".Alarma_On )
      Coil( "DB_SUB_1_GENERAL".Concatenadoras[13] )
   END_RUNG
   RUNG wire#powerrail
      Contact( "DB_SUB_1_GENERAL".Estados[23] )
      I_Contact( "01_LINEA_Entradas-DB".Canal3_Full )
      Contact( "01_LINEA_Entradas-DB".Canal1_Full )
   END_RUNG wire#w1
   // the same network as SCL:
   "DB_SUB_1_GENERAL".Concatenadoras[13] := (("DB_SUB_1_GENERAL".Estados[12] AND #DoneXN AND #DoneY) OR ("DB_SUB_1_GENERAL".Estados[23] AND NOT "01_LINEA_Entradas-DB".Canal3_Full AND "01_LINEA_Entradas-DB".Canal1_Full)) AND NOT "DB_INC_GENERAL".Alarma_On;
END_REGION

REGION Network 24: Concatenadora 14
   RUNG wire#powerrail
      Contact( "DB_SUB_1_GENERAL".Estados[13] )
      wire#w1
      Contact( #DoneYN )
      wire#w2
      Contact( "DB_SUB_1_GENERAL".Cuenta_1 )
      I_Contact( "DB_INC_GENERAL".Alarma_On )
      Coil( "DB_SUB_1_GENERAL".Concatenadoras[10] )
   END_RUNG
   RUNG wire#w1
      Contact( "Band_E23" )
   END_RUNG wire#w2
   // the same network as SCL:
   "DB_SUB_1_GENERAL".Concatenadoras[10] := "DB_SUB_1_GENERAL".Estados[13] AND (#DoneYN OR "Band_E23") AND "DB_SUB_1_GENERAL".Cuenta_1 AND NOT "DB_INC_GENERAL".Alarma_On;
END_REGION

REGION Network 25: Concatenadora 15
   RUNG wire#powerrail
      Contact( "DB_SUB_1_GENERAL".Estados[14] )
      wire#w1
      Contact( #Done2X )
      wire#w2
      Contact( #DoneY )
      wire#w3
      I_Contact( "DB_INC_GENERAL".Alarma_On )
      Coil( "DB_SUB_1_GENERAL".Concatenadoras[15] )
   END_RUNG
   RUNG wire#w1
      Contact( #DoneX )
   END_RUNG wire#w2
   RUNG wire#powerrail
      Contact( "DB_SUB_1_GENERAL".Estados[24] )
      I_Contact( "01_LINEA_Entradas-DB".Canal1_Full )
      Contact( "01_LINEA_Entradas-DB".Canal2_Full )
   END_RUNG wire#w3
   // the same network as SCL:
   "DB_SUB_1_GENERAL".Concatenadoras[15] := (("DB_SUB_1_GENERAL".Estados[14] AND (#Done2X OR #DoneX) AND #DoneY) OR ("DB_SUB_1_GENERAL".Estados[24] AND NOT "01_LINEA_Entradas-DB".Canal1_Full AND "01_LINEA_Entradas-DB".Canal2_Full)) AND NOT "DB_INC_GENERAL".Alarma_On;
END_REGION

REGION Network 26: Concatenadora 16
   RUNG wire#powerrail
      Contact( "DB_SUB_1_GENERAL".Estados[15] )
      wire#w1
      Contact( #DoneYN )
      wire#w2
      Contact( "DB_SUB_1_GENERAL".Cuenta_3 )
      I_Contact( "DB_INC_GENERAL".Alarma_On )
      Coil( "DB_SUB_1_GENERAL".Concatenadoras[16] )
   END_RUNG
   RUNG wire#w1
      Contact( "Band_E24" )
   END_RUNG wire#w2
   // the same network as SCL:
   "DB_SUB_1_GENERAL".Concatenadoras[16] := "DB_SUB_1_GENERAL".Estados[15] AND (#DoneYN OR "Band_E24") AND "DB_SUB_1_GENERAL".Cuenta_3 AND NOT "DB_INC_GENERAL".Alarma_On;
END_REGION

REGION Network 27: Concatenadora 17
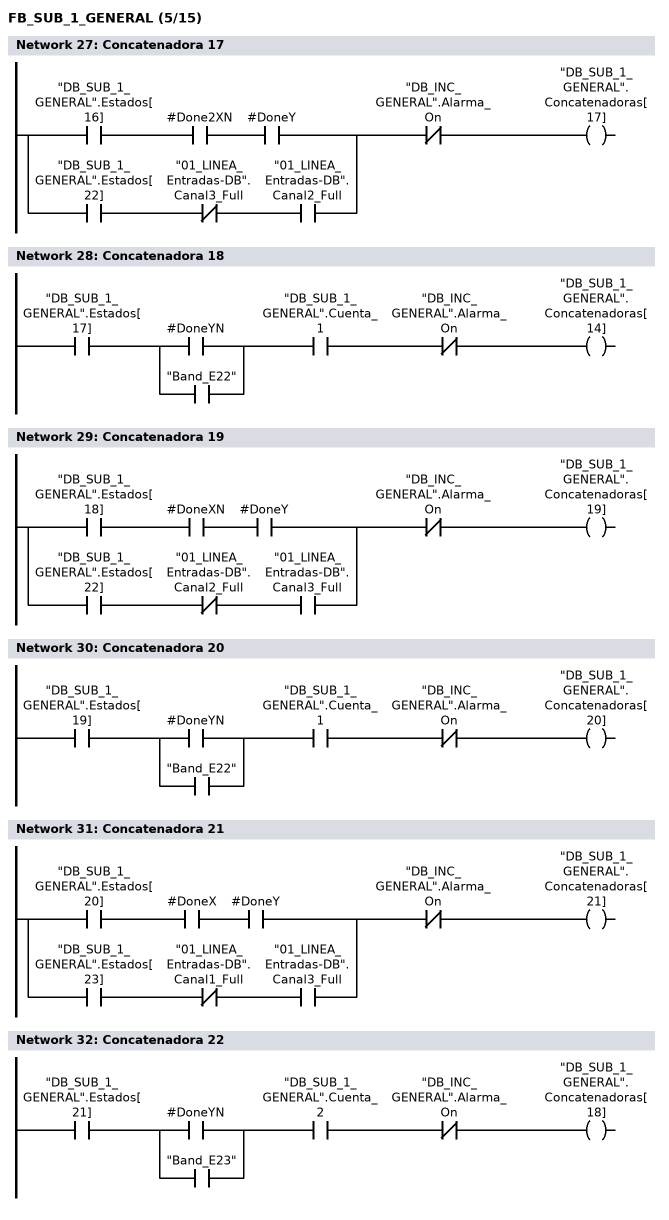
   RUNG wire#powerrail
      Contact( "DB_SUB_1_GENERAL".Estados[16] )
      Contact( #Done2XN )
      Contact( #DoneY )
      wire#w1
      I_Contact( "DB_INC_GENERAL".Alarma_On )
      Coil( "DB_SUB_1_GENERAL".Concatenadoras[17] )
   END_RUNG
   RUNG wire#powerrail
      Contact( "DB_SUB_1_GENERAL".Estados[22] )
      I_Contact( "01_LINEA_Entradas-DB".Canal3_Full )
      Contact( "01_LINEA_Entradas-DB".Canal2_Full )
   END_RUNG wire#w1
   // the same network as SCL:
   "DB_SUB_1_GENERAL".Concatenadoras[17] := (("DB_SUB_1_GENERAL".Estados[16] AND #Done2XN AND #DoneY) OR ("DB_SUB_1_GENERAL".Estados[22] AND NOT "01_LINEA_Entradas-DB".Canal3_Full AND "01_LINEA_Entradas-DB".Canal2_Full)) AND NOT "DB_INC_GENERAL".Alarma_On;
END_REGION

REGION Network 28: Concatenadora 18
   RUNG wire#powerrail
      Contact( "DB_SUB_1_GENERAL".Estados[17] )
      wire#w1
      Contact( #DoneYN )
      wire#w2
      Contact( "DB_SUB_1_GENERAL".Cuenta_1 )
      I_Contact( "DB_INC_GENERAL".Alarma_On )
      Coil( "DB_SUB_1_GENERAL".Concatenadoras[14] )
   END_RUNG
   RUNG wire#w1
      Contact( "Band_E22" )
   END_RUNG wire#w2
   // the same network as SCL:
   "DB_SUB_1_GENERAL".Concatenadoras[14] := "DB_SUB_1_GENERAL".Estados[17] AND (#DoneYN OR "Band_E22") AND "DB_SUB_1_GENERAL".Cuenta_1 AND NOT "DB_INC_GENERAL".Alarma_On;
END_REGION

REGION Network 29: Concatenadora 19
   RUNG wire#powerrail
      Contact( "DB_SUB_1_GENERAL".Estados[18] )
      Contact( #DoneXN )
      Contact( #DoneY )
      wire#w1
      I_Contact( "DB_INC_GENERAL".Alarma_On )
      Coil( "DB_SUB_1_GENERAL".Concatenadoras[19] )
   END_RUNG
   RUNG wire#powerrail
      Contact( "DB_SUB_1_GENERAL".Estados[22] )
      I_Contact( "01_LINEA_Entradas-DB".Canal2_Full )
      Contact( "01_LINEA_Entradas-DB".Canal3_Full )
   END_RUNG wire#w1
   // the same network as SCL:
   "DB_SUB_1_GENERAL".Concatenadoras[19] := (("DB_SUB_1_GENERAL".Estados[18] AND #DoneXN AND #DoneY) OR ("DB_SUB_1_GENERAL".Estados[22] AND NOT "01_LINEA_Entradas-DB".Canal2_Full AND "01_LINEA_Entradas-DB".Canal3_Full)) AND NOT "DB_INC_GENERAL".Alarma_On;
END_REGION

REGION Network 30: Concatenadora 20
   RUNG wire#powerrail
      Contact( "DB_SUB_1_GENERAL".Estados[19] )
      wire#w1
      Contact( #DoneYN )
      wire#w2
      Contact( "DB_SUB_1_GENERAL".Cuenta_1 )
      I_Contact( "DB_INC_GENERAL".Alarma_On )
      Coil( "DB_SUB_1_GENERAL".Concatenadoras[20] )
   END_RUNG
   RUNG wire#w1
      Contact( "Band_E22" )
   END_RUNG wire#w2
   // the same network as SCL:
   "DB_SUB_1_GENERAL".Concatenadoras[20] := "DB_SUB_1_GENERAL".Estados[19] AND (#DoneYN OR "Band_E22") AND "DB_SUB_1_GENERAL".Cuenta_1 AND NOT "DB_INC_GENERAL".Alarma_On;
END_REGION

REGION Network 31: Concatenadora 21
   RUNG wire#powerrail
      Contact( "DB_SUB_1_GENERAL".Estados[20] )
      Contact( #DoneX )
      Contact( #DoneY )
      wire#w1
      I_Contact( "DB_INC_GENERAL".Alarma_On )
      Coil( "DB_SUB_1_GENERAL".Concatenadoras[21] )
   END_RUNG
   RUNG wire#powerrail
      Contact( "DB_SUB_1_GENERAL".Estados[23] )
      I_Contact( "01_LINEA_Entradas-DB".Canal1_Full )
      Contact( "01_LINEA_Entradas-DB".Canal3_Full )
   END_RUNG wire#w1
   // the same network as SCL:
   "DB_SUB_1_GENERAL".Concatenadoras[21] := (("DB_SUB_1_GENERAL".Estados[20] AND #DoneX AND #DoneY) OR ("DB_SUB_1_GENERAL".Estados[23] AND NOT "01_LINEA_Entradas-DB".Canal1_Full AND "01_LINEA_Entradas-DB".Canal3_Full)) AND NOT "DB_INC_GENERAL".Alarma_On;
END_REGION

REGION Network 32: Concatenadora 22
   RUNG wire#powerrail
      Contact( "DB_SUB_1_GENERAL".Estados[21] )
      wire#w1
      Contact( #DoneYN )
      wire#w2
      Contact( "DB_SUB_1_GENERAL".Cuenta_2 )
      I_Contact( "DB_INC_GENERAL".Alarma_On )
      Coil( "DB_SUB_1_GENERAL".Concatenadoras[18] )
   END_RUNG
   RUNG wire#w1
      Contact( "Band_E23" )
   END_RUNG wire#w2
   // the same network as SCL:
   "DB_SUB_1_GENERAL".Concatenadoras[18] := "DB_SUB_1_GENERAL".Estados[21] AND (#DoneYN OR "Band_E23") AND "DB_SUB_1_GENERAL".Cuenta_2 AND NOT "DB_INC_GENERAL".Alarma_On;
END_REGION

REGION Network 33: Prioritaria 0
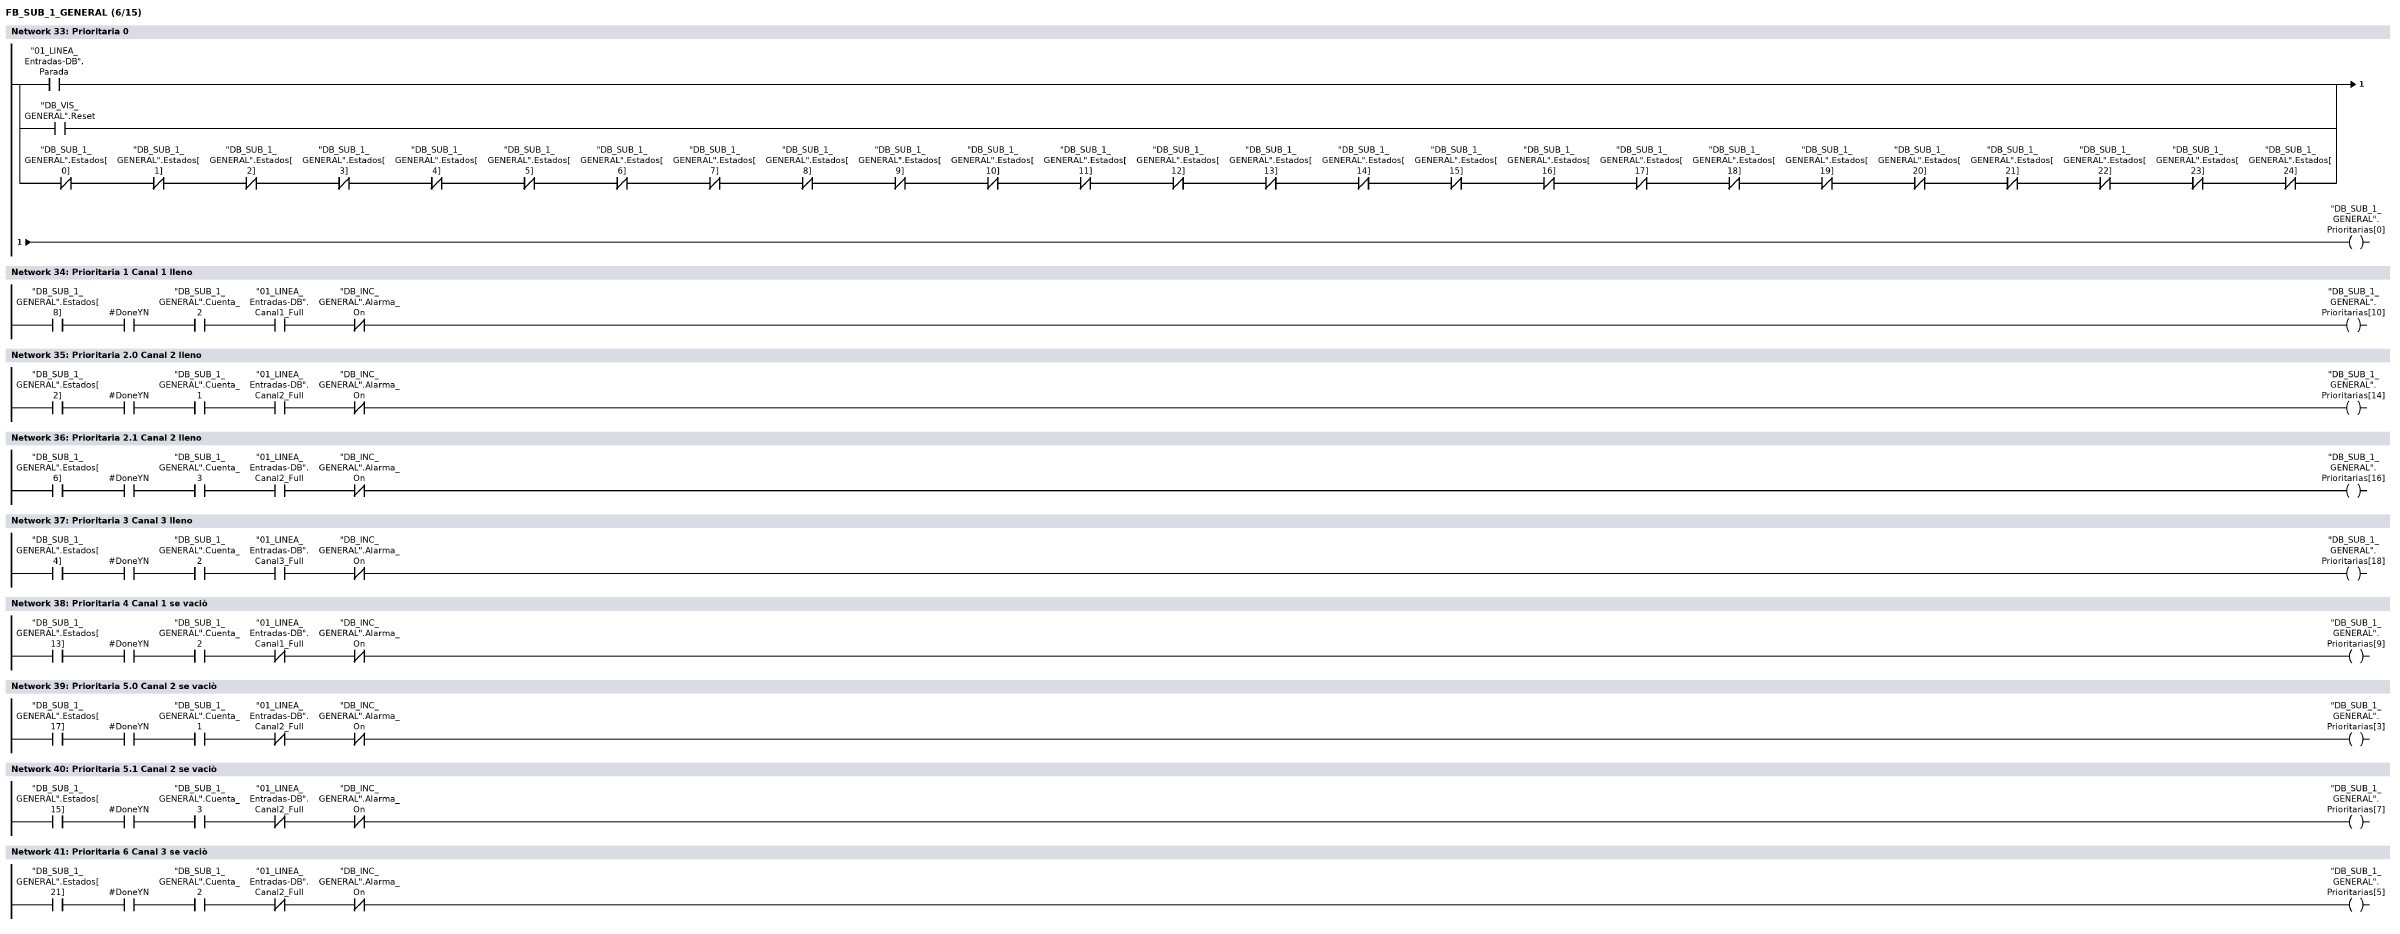
   RUNG wire#powerrail
      Contact( "01_LINEA_Entradas-DB".Parada )
      wire#w1
      Coil( "DB_SUB_1_GENERAL".Prioritarias[0] )
   END_RUNG
   RUNG wire#powerrail
      Contact( "DB_VIS_GENERAL".Reset )
   END_RUNG wire#w1
   RUNG wire#powerrail
      I_Contact( "DB_SUB_1_GENERAL".Estados[0] )
      I_Contact( "DB_SUB_1_GENERAL".Estados[1] )
      I_Contact( "DB_SUB_1_GENERAL".Estados[2] )
      I_Contact( "DB_SUB_1_GENERAL".Estados[3] )
      I_Contact( "DB_SUB_1_GENERAL".Estados[4] )
      I_Contact( "DB_SUB_1_GENERAL".Estados[5] )
      I_Contact( "DB_SUB_1_GENERAL".Estados[6] )
      I_Contact( "DB_SUB_1_GENERAL".Estados[7] )
      I_Contact( "DB_SUB_1_GENERAL".Estados[8] )
      I_Contact( "DB_SUB_1_GENERAL".Estados[9] )
      I_Contact( "DB_SUB_1_GENERAL".Estados[10] )
      I_Contact( "DB_SUB_1_GENERAL".Estados[11] )
      I_Contact( "DB_SUB_1_GENERAL".Estados[12] )
      I_Contact( "DB_SUB_1_GENERAL".Estados[13] )
      I_Contact( "DB_SUB_1_GENERAL".Estados[14] )
      I_Contact( "DB_SUB_1_GENERAL".Estados[15] )
      I_Contact( "DB_SUB_1_GENERAL".Estados[16] )
      I_Contact( "DB_SUB_1_GENERAL".Estados[17] )
      I_Contact( "DB_SUB_1_GENERAL".Estados[18] )
      I_Contact( "DB_SUB_1_GENERAL".Estados[19] )
      I_Contact( "DB_SUB_1_GENERAL".Estados[20] )
      I_Contact( "DB_SUB_1_GENERAL".Estados[21] )
      I_Contact( "DB_SUB_1_GENERAL".Estados[22] )
      I_Contact( "DB_SUB_1_GENERAL".Estados[23] )
      I_Contact( "DB_SUB_1_GENERAL".Estados[24] )
   END_RUNG wire#w1
   // the same network as SCL:
   "DB_SUB_1_GENERAL".Prioritarias[0] := "01_LINEA_Entradas-DB".Parada OR "DB_VIS_GENERAL".Reset OR (NOT "DB_SUB_1_GENERAL".Estados[0] AND NOT "DB_SUB_1_GENERAL".Estados[1] AND NOT "DB_SUB_1_GENERAL".Estados[2] AND NOT "DB_SUB_1_GENERAL".Estados[3] AND NOT "DB_SUB_1_GENERAL".Estados[4] AND NOT "DB_SUB_1_GENERAL".Estados[5] AND NOT "DB_SUB_1_GENERAL".Estados[6] AND NOT "DB_SUB_1_GENERAL".Estados[7] AND NOT "DB_SUB_1_GENERAL".Estados[8] AND NOT "DB_SUB_1_GENERAL".Estados[9] AND NOT "DB_SUB_1_GENERAL".Estados[10] AND NOT "DB_SUB_1_GENERAL".Estados[11] AND NOT "DB_SUB_1_GENERAL".Estados[12] AND NOT "DB_SUB_1_GENERAL".Estados[13] AND NOT "DB_SUB_1_GENERAL".Estados[14] AND NOT "DB_SUB_1_GENERAL".Estados[15] AND NOT "DB_SUB_1_GENERAL".Estados[16] AND NOT "DB_SUB_1_GENERAL".Estados[17] AND NOT "DB_SUB_1_GENERAL".Estados[18] AND NOT "DB_SUB_1_GENERAL".Estados[19] AND NOT "DB_SUB_1_GENERAL".Estados[20] AND NOT "DB_SUB_1_GENERAL".Estados[21] AND NOT "DB_SUB_1_GENERAL".Estados[22] AND NOT "DB_SUB_1_GENERAL".Estados[23] AND NOT "DB_SUB_1_GENERAL".Estados[24]);
END_REGION

REGION Network 34: Prioritaria 1 Canal 1 lleno
   RUNG wire#powerrail
      Contact( "DB_SUB_1_GENERAL".Estados[8] )
      Contact( #DoneYN )
      Contact( "DB_SUB_1_GENERAL".Cuenta_2 )
      Contact( "01_LINEA_Entradas-DB".Canal1_Full )
      I_Contact( "DB_INC_GENERAL".Alarma_On )
      Coil( "DB_SUB_1_GENERAL".Prioritarias[10] )
   END_RUNG
   // the same network as SCL:
   "DB_SUB_1_GENERAL".Prioritarias[10] := "DB_SUB_1_GENERAL".Estados[8] AND #DoneYN AND "DB_SUB_1_GENERAL".Cuenta_2 AND "01_LINEA_Entradas-DB".Canal1_Full AND NOT "DB_INC_GENERAL".Alarma_On;
END_REGION

REGION Network 35: Prioritaria 2.0 Canal 2 lleno
   RUNG wire#powerrail
      Contact( "DB_SUB_1_GENERAL".Estados[2] )
      Contact( #DoneYN )
      Contact( "DB_SUB_1_GENERAL".Cuenta_1 )
      Contact( "01_LINEA_Entradas-DB".Canal2_Full )
      I_Contact( "DB_INC_GENERAL".Alarma_On )
      Coil( "DB_SUB_1_GENERAL".Prioritarias[14] )
   END_RUNG
   // the same network as SCL:
   "DB_SUB_1_GENERAL".Prioritarias[14] := "DB_SUB_1_GENERAL".Estados[2] AND #DoneYN AND "DB_SUB_1_GENERAL".Cuenta_1 AND "01_LINEA_Entradas-DB".Canal2_Full AND NOT "DB_INC_GENERAL".Alarma_On;
END_REGION

REGION Network 36: Prioritaria 2.1 Canal 2 lleno
   RUNG wire#powerrail
      Contact( "DB_SUB_1_GENERAL".Estados[6] )
      Contact( #DoneYN )
      Contact( "DB_SUB_1_GENERAL".Cuenta_3 )
      Contact( "01_LINEA_Entradas-DB".Canal2_Full )
      I_Contact( "DB_INC_GENERAL".Alarma_On )
      Coil( "DB_SUB_1_GENERAL".Prioritarias[16] )
   END_RUNG
   // the same network as SCL:
   "DB_SUB_1_GENERAL".Prioritarias[16] := "DB_SUB_1_GENERAL".Estados[6] AND #DoneYN AND "DB_SUB_1_GENERAL".Cuenta_3 AND "01_LINEA_Entradas-DB".Canal2_Full AND NOT "DB_INC_GENERAL".Alarma_On;
END_REGION

REGION Network 37: Prioritaria 3 Canal 3 lleno
   RUNG wire#powerrail
      Contact( "DB_SUB_1_GENERAL".Estados[4] )
      Contact( #DoneYN )
      Contact( "DB_SUB_1_GENERAL".Cuenta_2 )
      Contact( "01_LINEA_Entradas-DB".Canal3_Full )
      I_Contact( "DB_INC_GENERAL".Alarma_On )
      Coil( "DB_SUB_1_GENERAL".Prioritarias[18] )
   END_RUNG
   // the same network as SCL:
   "DB_SUB_1_GENERAL".Prioritarias[18] := "DB_SUB_1_GENERAL".Estados[4] AND #DoneYN AND "DB_SUB_1_GENERAL".Cuenta_2 AND "01_LINEA_Entradas-DB".Canal3_Full AND NOT "DB_INC_GENERAL".Alarma_On;
END_REGION

REGION Network 38: Prioritaria 4 Canal 1 se vaciò
   RUNG wire#powerrail
      Contact( "DB_SUB_1_GENERAL".Estados[13] )
      Contact( #DoneYN )
      Contact( "DB_SUB_1_GENERAL".Cuenta_2 )
      I_Contact( "01_LINEA_Entradas-DB".Canal1_Full )
      I_Contact( "DB_INC_GENERAL".Alarma_On )
      Coil( "DB_SUB_1_GENERAL".Prioritarias[9] )
   END_RUNG
   // the same network as SCL:
   "DB_SUB_1_GENERAL".Prioritarias[9] := "DB_SUB_1_GENERAL".Estados[13] AND #DoneYN AND "DB_SUB_1_GENERAL".Cuenta_2 AND NOT "01_LINEA_Entradas-DB".Canal1_Full AND NOT "DB_INC_GENERAL".Alarma_On;
END_REGION

REGION Network 39: Prioritaria 5.0 Canal 2 se vaciò
   RUNG wire#powerrail
      Contact( "DB_SUB_1_GENERAL".Estados[17] )
      Contact( #DoneYN )
      Contact( "DB_SUB_1_GENERAL".Cuenta_1 )
      I_Contact( "01_LINEA_Entradas-DB".Canal2_Full )
      I_Contact( "DB_INC_GENERAL".Alarma_On )
      Coil( "DB_SUB_1_GENERAL".Prioritarias[3] )
   END_RUNG
   // the same network as SCL:
   "DB_SUB_1_GENERAL".Prioritarias[3] := "DB_SUB_1_GENERAL".Estados[17] AND #DoneYN AND "DB_SUB_1_GENERAL".Cuenta_1 AND NOT "01_LINEA_Entradas-DB".Canal2_Full AND NOT "DB_INC_GENERAL".Alarma_On;
END_REGION

REGION Network 40: Prioritaria 5.1 Canal 2 se vaciò
   RUNG wire#powerrail
      Contact( "DB_SUB_1_GENERAL".Estados[15] )
      Contact( #DoneYN )
      Contact( "DB_SUB_1_GENERAL".Cuenta_3 )
      I_Contact( "01_LINEA_Entradas-DB".Canal2_Full )
      I_Contact( "DB_INC_GENERAL".Alarma_On )
      Coil( "DB_SUB_1_GENERAL".Prioritarias[7] )
   END_RUNG
   // the same network as SCL:
   "DB_SUB_1_GENERAL".Prioritarias[7] := "DB_SUB_1_GENERAL".Estados[15] AND #DoneYN AND "DB_SUB_1_GENERAL".Cuenta_3 AND NOT "01_LINEA_Entradas-DB".Canal2_Full AND NOT "DB_INC_GENERAL".Alarma_On;
END_REGION

REGION Network 41: Prioritaria 6 Canal 3 se vaciò
   RUNG wire#powerrail
      Contact( "DB_SUB_1_GENERAL".Estados[21] )
      Contact( #DoneYN )
      Contact( "DB_SUB_1_GENERAL".Cuenta_2 )
      I_Contact( "01_LINEA_Entradas-DB".Canal2_Full )
      I_Contact( "DB_INC_GENERAL".Alarma_On )
      Coil( "DB_SUB_1_GENERAL".Prioritarias[5] )
   END_RUNG
   // the same network as SCL:
   "DB_SUB_1_GENERAL".Prioritarias[5] := "DB_SUB_1_GENERAL".Estados[21] AND #DoneYN AND "DB_SUB_1_GENERAL".Cuenta_2 AND NOT "01_LINEA_Entradas-DB".Canal2_Full AND NOT "DB_INC_GENERAL".Alarma_On;
END_REGION

REGION Network 42: Prioritaria 7 Canal 2 y 3 llenos
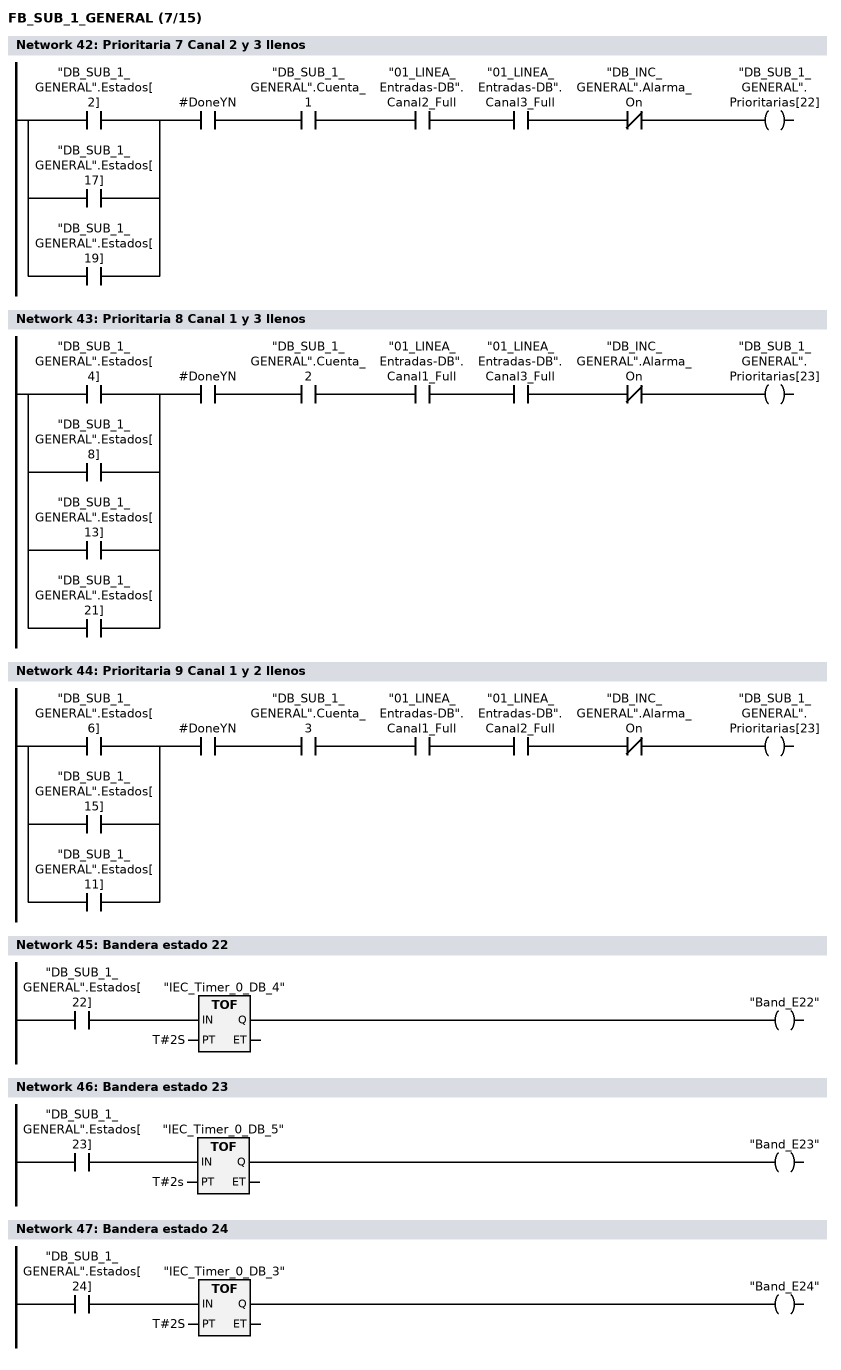
   RUNG wire#powerrail
      Contact( "DB_SUB_1_GENERAL".Estados[2] )
      wire#w1
      Contact( #DoneYN )
      Contact( "DB_SUB_1_GENERAL".Cuenta_1 )
      Contact( "01_LINEA_Entradas-DB".Canal2_Full )
      Contact( "01_LINEA_Entradas-DB".Canal3_Full )
      I_Contact( "DB_INC_GENERAL".Alarma_On )
      Coil( "DB_SUB_1_GENERAL".Prioritarias[22] )
   END_RUNG
   RUNG wire#powerrail
      Contact( "DB_SUB_1_GENERAL".Estados[17] )
   END_RUNG wire#w1
   RUNG wire#powerrail
      Contact( "DB_SUB_1_GENERAL".Estados[19] )
   END_RUNG wire#w1
   // the same network as SCL:
   "DB_SUB_1_GENERAL".Prioritarias[22] := ("DB_SUB_1_GENERAL".Estados[2] OR "DB_SUB_1_GENERAL".Estados[17] OR "DB_SUB_1_GENERAL".Estados[19]) AND #DoneYN AND "DB_SUB_1_GENERAL".Cuenta_1 AND "01_LINEA_Entradas-DB".Canal2_Full AND "01_LINEA_Entradas-DB".Canal3_Full AND NOT "DB_INC_GENERAL".Alarma_On;
END_REGION

REGION Network 43: Prioritaria 8 Canal 1 y 3 llenos
   RUNG wire#powerrail
      Contact( "DB_SUB_1_GENERAL".Estados[4] )
      wire#w1
      Contact( #DoneYN )
      Contact( "DB_SUB_1_GENERAL".Cuenta_2 )
      Contact( "01_LINEA_Entradas-DB".Canal1_Full )
      Contact( "01_LINEA_Entradas-DB".Canal3_Full )
      I_Contact( "DB_INC_GENERAL".Alarma_On )
      Coil( "DB_SUB_1_GENERAL".Prioritarias[23] )
   END_RUNG
   RUNG wire#powerrail
      Contact( "DB_SUB_1_GENERAL".Estados[8] )
   END_RUNG wire#w1
   RUNG wire#powerrail
      Contact( "DB_SUB_1_GENERAL".Estados[13] )
   END_RUNG wire#w1
   RUNG wire#powerrail
      Contact( "DB_SUB_1_GENERAL".Estados[21] )
   END_RUNG wire#w1
   // the same network as SCL:
   "DB_SUB_1_GENERAL".Prioritarias[23] := ("DB_SUB_1_GENERAL".Estados[4] OR "DB_SUB_1_GENERAL".Estados[8] OR "DB_SUB_1_GENERAL".Estados[13] OR "DB_SUB_1_GENERAL".Estados[21]) AND #DoneYN AND "DB_SUB_1_GENERAL".Cuenta_2 AND "01_LINEA_Entradas-DB".Canal1_Full AND "01_LINEA_Entradas-DB".Canal3_Full AND NOT "DB_INC_GENERAL".Alarma_On;
END_REGION

REGION Network 44: Prioritaria 9 Canal 1 y 2 llenos
   RUNG wire#powerrail
      Contact( "DB_SUB_1_GENERAL".Estados[6] )
      wire#w1
      Contact( #DoneYN )
      Contact( "DB_SUB_1_GENERAL".Cuenta_3 )
      Contact( "01_LINEA_Entradas-DB".Canal1_Full )
      Contact( "01_LINEA_Entradas-DB".Canal2_Full )
      I_Contact( "DB_INC_GENERAL".Alarma_On )
      Coil( "DB_SUB_1_GENERAL".Prioritarias[23] )
   END_RUNG
   RUNG wire#powerrail
      Contact( "DB_SUB_1_GENERAL".Estados[15] )
   END_RUNG wire#w1
   RUNG wire#powerrail
      Contact( "DB_SUB_1_GENERAL".Estados[11] )
   END_RUNG wire#w1
   // the same network as SCL:
   "DB_SUB_1_GENERAL".Prioritarias[23] := ("DB_SUB_1_GENERAL".Estados[6] OR "DB_SUB_1_GENERAL".Estados[15] OR "DB_SUB_1_GENERAL".Estados[11]) AND #DoneYN AND "DB_SUB_1_GENERAL".Cuenta_3 AND "01_LINEA_Entradas-DB".Canal1_Full AND "01_LINEA_Entradas-DB".Canal2_Full AND NOT "DB_INC_GENERAL".Alarma_On;
END_REGION

REGION Network 45: Bandera estado 22
   "IEC_Timer_0_DB_4".TOF(IN := "DB_SUB_1_GENERAL".Estados[22], PT := T#2S);
   "Band_E22" := "IEC_Timer_0_DB_4".Q;
END_REGION

REGION Network 46: Bandera estado 23
   "IEC_Timer_0_DB_5".TOF(IN := "DB_SUB_1_GENERAL".Estados[23], PT := T#2s);
   "Band_E23" := "IEC_Timer_0_DB_5".Q;
END_REGION

REGION Network 47: Bandera estado 24
   "IEC_Timer_0_DB_3".TOF(IN := "DB_SUB_1_GENERAL".Estados[24], PT := T#2S);
   "Band_E24" := "IEC_Timer_0_DB_3".Q;
END_REGION

REGION Network 48: BLOQUE MAQUINA ESTADO
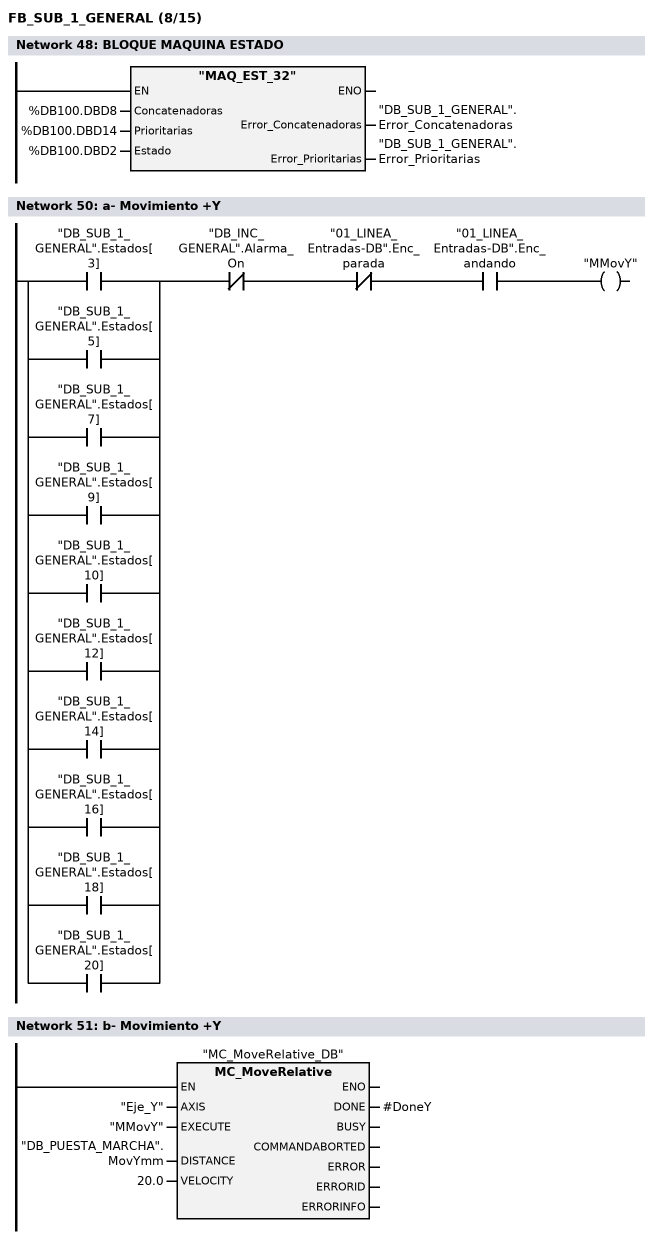
   RUNG wire#powerrail
      "MAQ_EST_32"(Concatenadoras := %DB100.DBD8, Prioritarias := %DB100.DBD14, Estado := %DB100.DBD2, Error_Concatenadoras => "DB_SUB_1_GENERAL".Error_Concatenadoras, Error_Prioritarias => "DB_SUB_1_GENERAL".Error_Prioritarias)
   END_RUNG
   // the same network as SCL:
   "MAQ_EST_32"(Concatenadoras := %DB100.DBD8,
                Prioritarias := %DB100.DBD14,
                Estado := %DB100.DBD2,
                Error_Concatenadoras => "DB_SUB_1_GENERAL".Error_Concatenadoras,
                Error_Prioritarias => "DB_SUB_1_GENERAL".Error_Prioritarias);
END_REGION

REGION Network 49: --------------ACCIONAMIENTOS----------------
END_REGION

REGION Network 50: a- Movimiento +Y
   RUNG wire#powerrail
      Contact( "DB_SUB_1_GENERAL".Estados[3] )
      wire#w1
      I_Contact( "DB_INC_GENERAL".Alarma_On )
      I_Contact( "01_LINEA_Entradas-DB".Enc_parada )
      Contact( "01_LINEA_Entradas-DB".Enc_andando )
      Coil( "MMovY" )
   END_RUNG
   RUNG wire#powerrail
      Contact( "DB_SUB_1_GENERAL".Estados[5] )
   END_RUNG wire#w1
   RUNG wire#powerrail
      Contact( "DB_SUB_1_GENERAL".Estados[7] )
   END_RUNG wire#w1
   RUNG wire#powerrail
      Contact( "DB_SUB_1_GENERAL".Estados[9] )
   END_RUNG wire#w1
   RUNG wire#powerrail
      Contact( "DB_SUB_1_GENERAL".Estados[10] )
   END_RUNG wire#w1
   RUNG wire#powerrail
      Contact( "DB_SUB_1_GENERAL".Estados[12] )
   END_RUNG wire#w1
   RUNG wire#powerrail
      Contact( "DB_SUB_1_GENERAL".Estados[14] )
   END_RUNG wire#w1
   RUNG wire#powerrail
      Contact( "DB_SUB_1_GENERAL".Estados[16] )
   END_RUNG wire#w1
   RUNG wire#powerrail
      Contact( "DB_SUB_1_GENERAL".Estados[18] )
   END_RUNG wire#w1
   RUNG wire#powerrail
      Contact( "DB_SUB_1_GENERAL".Estados[20] )
   END_RUNG wire#w1
   // the same network as SCL:
   "MMovY" := ("DB_SUB_1_GENERAL".Estados[3] OR "DB_SUB_1_GENERAL".Estados[5] OR "DB_SUB_1_GENERAL".Estados[7] OR "DB_SUB_1_GENERAL".Estados[9] OR "DB_SUB_1_GENERAL".Estados[10] OR "DB_SUB_1_GENERAL".Estados[12] OR "DB_SUB_1_GENERAL".Estados[14] OR "DB_SUB_1_GENERAL".Estados[16] OR "DB_SUB_1_GENERAL".Estados[18] OR "DB_SUB_1_GENERAL".Estados[20]) AND NOT "DB_INC_GENERAL".Alarma_On AND NOT "01_LINEA_Entradas-DB".Enc_parada AND "01_LINEA_Entradas-DB".Enc_andando;
END_REGION

REGION Network 51: b- Movimiento +Y
   "MC_MoveRelative_DB"(Axis := "Eje_Y",   // MC_MoveRelative
                        Execute := "MMovY",
                        Distance := "DB_PUESTA_MARCHA".MovYmm,
                        Velocity := 20.0,
                        Done => #DoneY);
END_REGION

REGION Network 52: a- Movimiento -Y
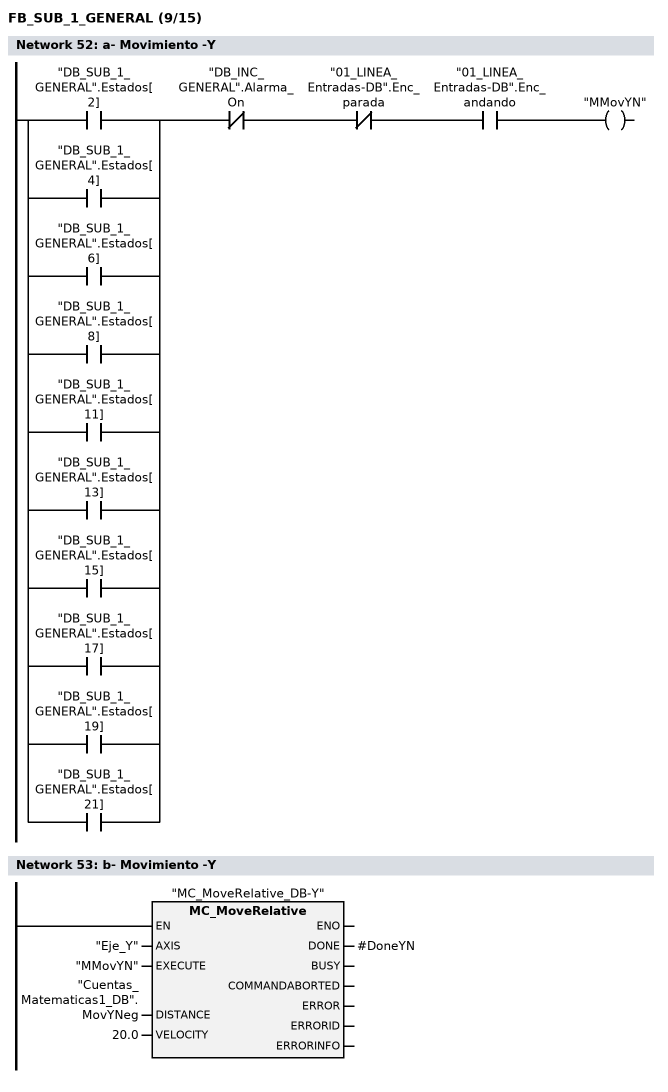
   RUNG wire#powerrail
      Contact( "DB_SUB_1_GENERAL".Estados[2] )
      wire#w1
      I_Contact( "DB_INC_GENERAL".Alarma_On )
      I_Contact( "01_LINEA_Entradas-DB".Enc_parada )
      Contact( "01_LINEA_Entradas-DB".Enc_andando )
      Coil( "MMovYN" )
   END_RUNG
   RUNG wire#powerrail
      Contact( "DB_SUB_1_GENERAL".Estados[4] )
   END_RUNG wire#w1
   RUNG wire#powerrail
      Contact( "DB_SUB_1_GENERAL".Estados[6] )
   END_RUNG wire#w1
   RUNG wire#powerrail
      Contact( "DB_SUB_1_GENERAL".Estados[8] )
   END_RUNG wire#w1
   RUNG wire#powerrail
      Contact( "DB_SUB_1_GENERAL".Estados[11] )
   END_RUNG wire#w1
   RUNG wire#powerrail
      Contact( "DB_SUB_1_GENERAL".Estados[13] )
   END_RUNG wire#w1
   RUNG wire#powerrail
      Contact( "DB_SUB_1_GENERAL".Estados[15] )
   END_RUNG wire#w1
   RUNG wire#powerrail
      Contact( "DB_SUB_1_GENERAL".Estados[17] )
   END_RUNG wire#w1
   RUNG wire#powerrail
      Contact( "DB_SUB_1_GENERAL".Estados[19] )
   END_RUNG wire#w1
   RUNG wire#powerrail
      Contact( "DB_SUB_1_GENERAL".Estados[21] )
   END_RUNG wire#w1
   // the same network as SCL:
   "MMovYN" := ("DB_SUB_1_GENERAL".Estados[2] OR "DB_SUB_1_GENERAL".Estados[4] OR "DB_SUB_1_GENERAL".Estados[6] OR "DB_SUB_1_GENERAL".Estados[8] OR "DB_SUB_1_GENERAL".Estados[11] OR "DB_SUB_1_GENERAL".Estados[13] OR "DB_SUB_1_GENERAL".Estados[15] OR "DB_SUB_1_GENERAL".Estados[17] OR "DB_SUB_1_GENERAL".Estados[19] OR "DB_SUB_1_GENERAL".Estados[21]) AND NOT "DB_INC_GENERAL".Alarma_On AND NOT "01_LINEA_Entradas-DB".Enc_parada AND "01_LINEA_Entradas-DB".Enc_andando;
END_REGION

REGION Network 53: b- Movimiento -Y
   "MC_MoveRelative_DB-Y"(Axis := "Eje_Y",   // MC_MoveRelative
                          Execute := "MMovYN",
                          Distance := "Cuentas_Matematicas1_DB".MovYNeg,
                          Velocity := 20.0,
                          Done => #DoneYN);
END_REGION

REGION Network 54: a- Movimiento +X
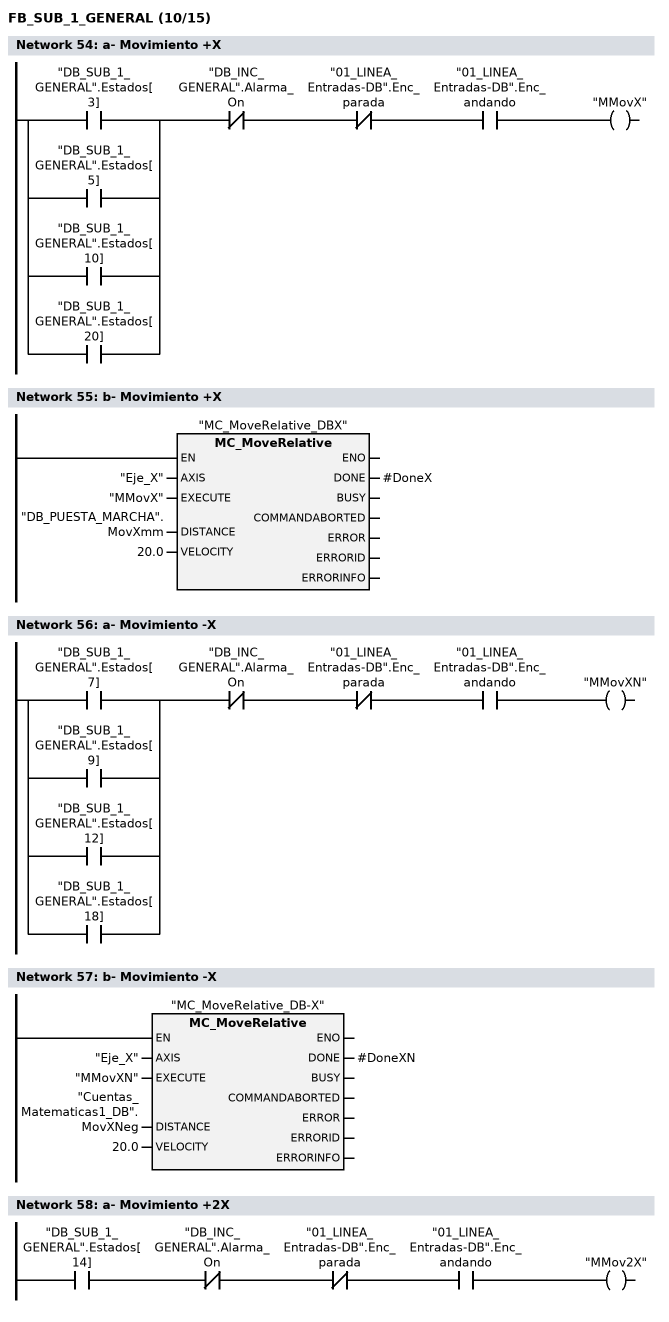
   RUNG wire#powerrail
      Contact( "DB_SUB_1_GENERAL".Estados[3] )
      wire#w1
      I_Contact( "DB_INC_GENERAL".Alarma_On )
      I_Contact( "01_LINEA_Entradas-DB".Enc_parada )
      Contact( "01_LINEA_Entradas-DB".Enc_andando )
      Coil( "MMovX" )
   END_RUNG
   RUNG wire#powerrail
      Contact( "DB_SUB_1_GENERAL".Estados[5] )
   END_RUNG wire#w1
   RUNG wire#powerrail
      Contact( "DB_SUB_1_GENERAL".Estados[10] )
   END_RUNG wire#w1
   RUNG wire#powerrail
      Contact( "DB_SUB_1_GENERAL".Estados[20] )
   END_RUNG wire#w1
   // the same network as SCL:
   "MMovX" := ("DB_SUB_1_GENERAL".Estados[3] OR "DB_SUB_1_GENERAL".Estados[5] OR "DB_SUB_1_GENERAL".Estados[10] OR "DB_SUB_1_GENERAL".Estados[20]) AND NOT "DB_INC_GENERAL".Alarma_On AND NOT "01_LINEA_Entradas-DB".Enc_parada AND "01_LINEA_Entradas-DB".Enc_andando;
END_REGION

REGION Network 55: b- Movimiento +X
   "MC_MoveRelative_DBX"(Axis := "Eje_X",   // MC_MoveRelative
                         Execute := "MMovX",
                         Distance := "DB_PUESTA_MARCHA".MovXmm,
                         Velocity := 20.0,
                         Done => #DoneX);
END_REGION

REGION Network 56: a- Movimiento -X
   RUNG wire#powerrail
      Contact( "DB_SUB_1_GENERAL".Estados[7] )
      wire#w1
      I_Contact( "DB_INC_GENERAL".Alarma_On )
      I_Contact( "01_LINEA_Entradas-DB".Enc_parada )
      Contact( "01_LINEA_Entradas-DB".Enc_andando )
      Coil( "MMovXN" )
   END_RUNG
   RUNG wire#powerrail
      Contact( "DB_SUB_1_GENERAL".Estados[9] )
   END_RUNG wire#w1
   RUNG wire#powerrail
      Contact( "DB_SUB_1_GENERAL".Estados[12] )
   END_RUNG wire#w1
   RUNG wire#powerrail
      Contact( "DB_SUB_1_GENERAL".Estados[18] )
   END_RUNG wire#w1
   // the same network as SCL:
   "MMovXN" := ("DB_SUB_1_GENERAL".Estados[7] OR "DB_SUB_1_GENERAL".Estados[9] OR "DB_SUB_1_GENERAL".Estados[12] OR "DB_SUB_1_GENERAL".Estados[18]) AND NOT "DB_INC_GENERAL".Alarma_On AND NOT "01_LINEA_Entradas-DB".Enc_parada AND "01_LINEA_Entradas-DB".Enc_andando;
END_REGION

REGION Network 57: b- Movimiento -X
   "MC_MoveRelative_DB-X"(Axis := "Eje_X",   // MC_MoveRelative
                          Execute := "MMovXN",
                          Distance := "Cuentas_Matematicas1_DB".MovXNeg,
                          Velocity := 20.0,
                          Done => #DoneXN);
END_REGION

REGION Network 58: a- Movimiento +2X
   RUNG wire#powerrail
      Contact( "DB_SUB_1_GENERAL".Estados[14] )
      I_Contact( "DB_INC_GENERAL".Alarma_On )
      I_Contact( "01_LINEA_Entradas-DB".Enc_parada )
      Contact( "01_LINEA_Entradas-DB".Enc_andando )
      Coil( "MMov2X" )
   END_RUNG
   // the same network as SCL:
   "MMov2X" := "DB_SUB_1_GENERAL".Estados[14] AND NOT "DB_INC_GENERAL".Alarma_On AND NOT "01_LINEA_Entradas-DB".Enc_parada AND "01_LINEA_Entradas-DB".Enc_andando;
END_REGION

REGION Network 59: b- Movimiento +2X
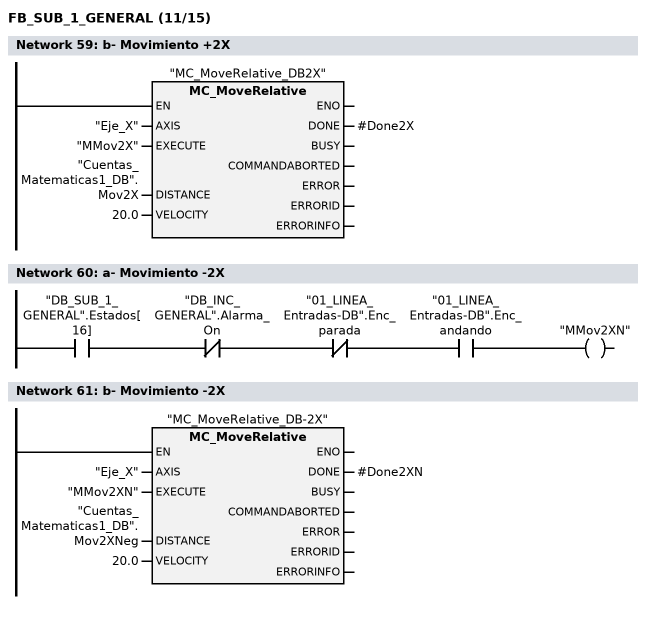
   "MC_MoveRelative_DB2X"(Axis := "Eje_X",   // MC_MoveRelative
                          Execute := "MMov2X",
                          Distance := "Cuentas_Matematicas1_DB".Mov2X,
                          Velocity := 20.0,
                          Done => #Done2X);
END_REGION

REGION Network 60: a- Movimiento -2X
   RUNG wire#powerrail
      Contact( "DB_SUB_1_GENERAL".Estados[16] )
      I_Contact( "DB_INC_GENERAL".Alarma_On )
      I_Contact( "01_LINEA_Entradas-DB".Enc_parada )
      Contact( "01_LINEA_Entradas-DB".Enc_andando )
      Coil( "MMov2XN" )
   END_RUNG
   // the same network as SCL:
   "MMov2XN" := "DB_SUB_1_GENERAL".Estados[16] AND NOT "DB_INC_GENERAL".Alarma_On AND NOT "01_LINEA_Entradas-DB".Enc_parada AND "01_LINEA_Entradas-DB".Enc_andando;
END_REGION

REGION Network 61: b- Movimiento -2X
   "MC_MoveRelative_DB-2X"(Axis := "Eje_X",   // MC_MoveRelative
                           Execute := "MMov2XN",
                           Distance := "Cuentas_Matematicas1_DB".Mov2XNeg,
                           Velocity := 20.0,
                           Done => #Done2XN);
END_REGION

REGION Network 62: Avance inverter
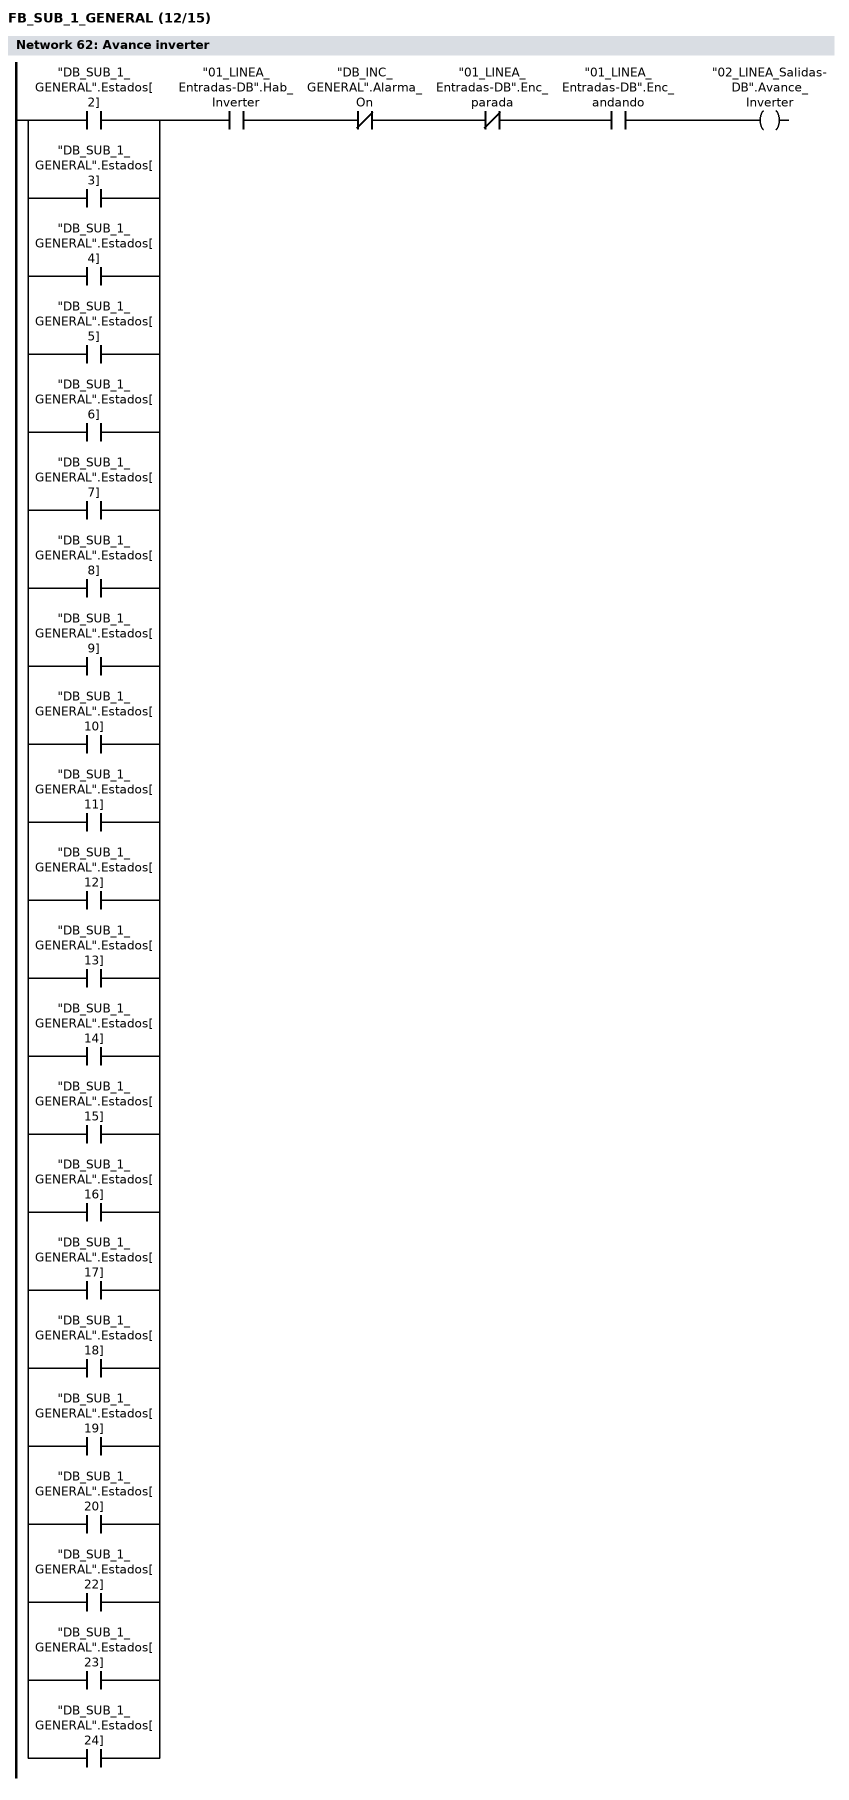
   RUNG wire#powerrail
      Contact( "DB_SUB_1_GENERAL".Estados[2] )
      wire#w1
      Contact( "01_LINEA_Entradas-DB".Hab_Inverter )
      I_Contact( "DB_INC_GENERAL".Alarma_On )
      I_Contact( "01_LINEA_Entradas-DB".Enc_parada )
      Contact( "01_LINEA_Entradas-DB".Enc_andando )
      Coil( "02_LINEA_Salidas-DB".Avance_Inverter )
   END_RUNG
   RUNG wire#powerrail
      Contact( "DB_SUB_1_GENERAL".Estados[3] )
   END_RUNG wire#w1
   RUNG wire#powerrail
      Contact( "DB_SUB_1_GENERAL".Estados[4] )
   END_RUNG wire#w1
   RUNG wire#powerrail
      Contact( "DB_SUB_1_GENERAL".Estados[5] )
   END_RUNG wire#w1
   RUNG wire#powerrail
      Contact( "DB_SUB_1_GENERAL".Estados[6] )
   END_RUNG wire#w1
   RUNG wire#powerrail
      Contact( "DB_SUB_1_GENERAL".Estados[7] )
   END_RUNG wire#w1
   RUNG wire#powerrail
      Contact( "DB_SUB_1_GENERAL".Estados[8] )
   END_RUNG wire#w1
   RUNG wire#powerrail
      Contact( "DB_SUB_1_GENERAL".Estados[9] )
   END_RUNG wire#w1
   RUNG wire#powerrail
      Contact( "DB_SUB_1_GENERAL".Estados[10] )
   END_RUNG wire#w1
   RUNG wire#powerrail
      Contact( "DB_SUB_1_GENERAL".Estados[11] )
   END_RUNG wire#w1
   RUNG wire#powerrail
      Contact( "DB_SUB_1_GENERAL".Estados[12] )
   END_RUNG wire#w1
   RUNG wire#powerrail
      Contact( "DB_SUB_1_GENERAL".Estados[13] )
   END_RUNG wire#w1
   RUNG wire#powerrail
      Contact( "DB_SUB_1_GENERAL".Estados[14] )
   END_RUNG wire#w1
   RUNG wire#powerrail
      Contact( "DB_SUB_1_GENERAL".Estados[15] )
   END_RUNG wire#w1
   RUNG wire#powerrail
      Contact( "DB_SUB_1_GENERAL".Estados[16] )
   END_RUNG wire#w1
   RUNG wire#powerrail
      Contact( "DB_SUB_1_GENERAL".Estados[17] )
   END_RUNG wire#w1
   RUNG wire#powerrail
      Contact( "DB_SUB_1_GENERAL".Estados[18] )
   END_RUNG wire#w1
   RUNG wire#powerrail
      Contact( "DB_SUB_1_GENERAL".Estados[19] )
   END_RUNG wire#w1
   RUNG wire#powerrail
      Contact( "DB_SUB_1_GENERAL".Estados[20] )
   END_RUNG wire#w1
   RUNG wire#powerrail
      Contact( "DB_SUB_1_GENERAL".Estados[22] )
   END_RUNG wire#w1
   RUNG wire#powerrail
      Contact( "DB_SUB_1_GENERAL".Estados[23] )
   END_RUNG wire#w1
   RUNG wire#powerrail
      Contact( "DB_SUB_1_GENERAL".Estados[24] )
   END_RUNG wire#w1
   // the same network as SCL:
   "02_LINEA_Salidas-DB".Avance_Inverter := ("DB_SUB_1_GENERAL".Estados[2] OR "DB_SUB_1_GENERAL".Estados[3] OR "DB_SUB_1_GENERAL".Estados[4] OR "DB_SUB_1_GENERAL".Estados[5] OR "DB_SUB_1_GENERAL".Estados[6] OR "DB_SUB_1_GENERAL".Estados[7] OR "DB_SUB_1_GENERAL".Estados[8] OR "DB_SUB_1_GENERAL".Estados[9] OR "DB_SUB_1_GENERAL".Estados[10] OR "DB_SUB_1_GENERAL".Estados[11] OR "DB_SUB_1_GENERAL".Estados[12] OR "DB_SUB_1_GENERAL".Estados[13] OR "DB_SUB_1_GENERAL".Estados[14] OR "DB_SUB_1_GENERAL".Estados[15] OR "DB_SUB_1_GENERAL".Estados[16] OR "DB_SUB_1_GENERAL".Estados[17] OR "DB_SUB_1_GENERAL".Estados[18] OR "DB_SUB_1_GENERAL".Estados[19] OR "DB_SUB_1_GENERAL".Estados[20] OR "DB_SUB_1_GENERAL".Estados[22] OR "DB_SUB_1_GENERAL".Estados[23] OR "DB_SUB_1_GENERAL".Estados[24]) AND "01_LINEA_Entradas-DB".Hab_Inverter AND NOT "DB_INC_GENERAL".Alarma_On AND NOT "01_LINEA_Entradas-DB".Enc_parada AND "01_LINEA_Entradas-DB".Enc_andando;
END_REGION

REGION Network 63: Divider en marcha
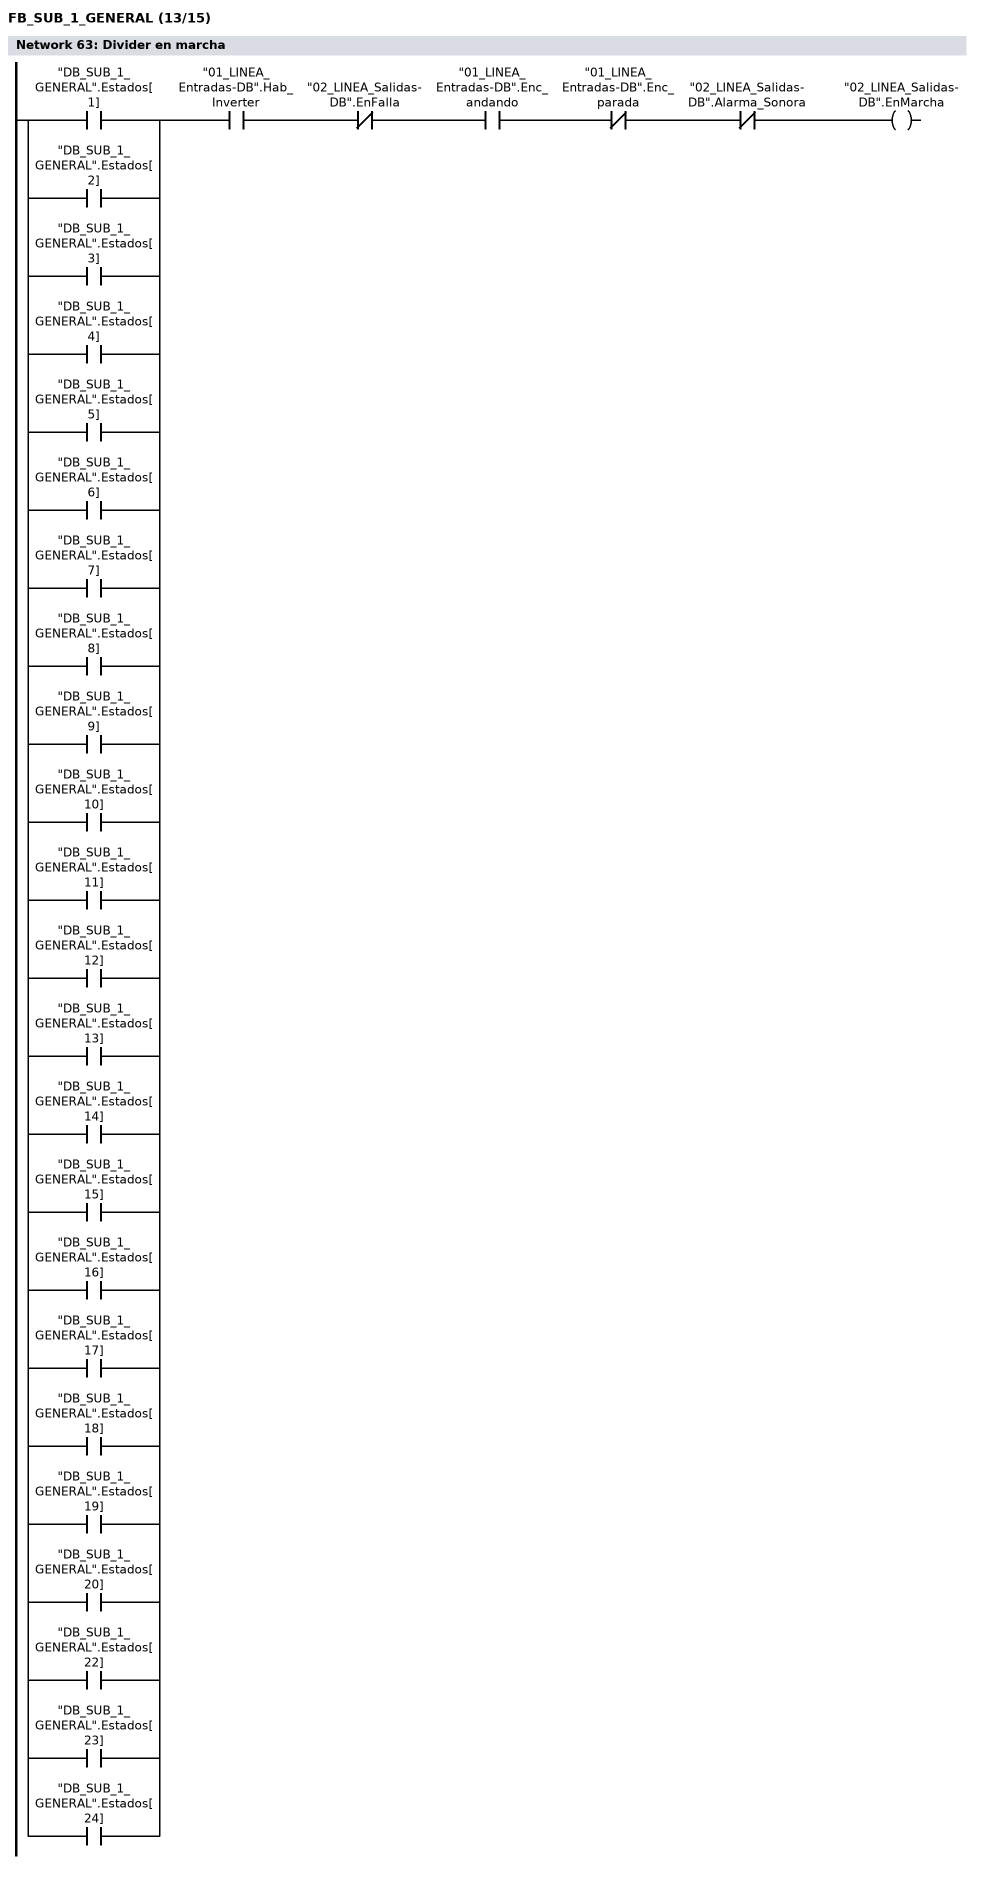
   RUNG wire#powerrail
      Contact( "DB_SUB_1_GENERAL".Estados[1] )
      wire#w1
      Contact( "01_LINEA_Entradas-DB".Hab_Inverter )
      I_Contact( "02_LINEA_Salidas-DB".EnFalla )
      Contact( "01_LINEA_Entradas-DB".Enc_andando )
      I_Contact( "01_LINEA_Entradas-DB".Enc_parada )
      I_Contact( "02_LINEA_Salidas-DB".Alarma_Sonora )
      Coil( "02_LINEA_Salidas-DB".EnMarcha )
   END_RUNG
   RUNG wire#powerrail
      Contact( "DB_SUB_1_GENERAL".Estados[2] )
   END_RUNG wire#w1
   RUNG wire#powerrail
      Contact( "DB_SUB_1_GENERAL".Estados[3] )
   END_RUNG wire#w1
   RUNG wire#powerrail
      Contact( "DB_SUB_1_GENERAL".Estados[4] )
   END_RUNG wire#w1
   RUNG wire#powerrail
      Contact( "DB_SUB_1_GENERAL".Estados[5] )
   END_RUNG wire#w1
   RUNG wire#powerrail
      Contact( "DB_SUB_1_GENERAL".Estados[6] )
   END_RUNG wire#w1
   RUNG wire#powerrail
      Contact( "DB_SUB_1_GENERAL".Estados[7] )
   END_RUNG wire#w1
   RUNG wire#powerrail
      Contact( "DB_SUB_1_GENERAL".Estados[8] )
   END_RUNG wire#w1
   RUNG wire#powerrail
      Contact( "DB_SUB_1_GENERAL".Estados[9] )
   END_RUNG wire#w1
   RUNG wire#powerrail
      Contact( "DB_SUB_1_GENERAL".Estados[10] )
   END_RUNG wire#w1
   RUNG wire#powerrail
      Contact( "DB_SUB_1_GENERAL".Estados[11] )
   END_RUNG wire#w1
   RUNG wire#powerrail
      Contact( "DB_SUB_1_GENERAL".Estados[12] )
   END_RUNG wire#w1
   RUNG wire#powerrail
      Contact( "DB_SUB_1_GENERAL".Estados[13] )
   END_RUNG wire#w1
   RUNG wire#powerrail
      Contact( "DB_SUB_1_GENERAL".Estados[14] )
   END_RUNG wire#w1
   RUNG wire#powerrail
      Contact( "DB_SUB_1_GENERAL".Estados[15] )
   END_RUNG wire#w1
   RUNG wire#powerrail
      Contact( "DB_SUB_1_GENERAL".Estados[16] )
   END_RUNG wire#w1
   RUNG wire#powerrail
      Contact( "DB_SUB_1_GENERAL".Estados[17] )
   END_RUNG wire#w1
   RUNG wire#powerrail
      Contact( "DB_SUB_1_GENERAL".Estados[18] )
   END_RUNG wire#w1
   RUNG wire#powerrail
      Contact( "DB_SUB_1_GENERAL".Estados[19] )
   END_RUNG wire#w1
   RUNG wire#powerrail
      Contact( "DB_SUB_1_GENERAL".Estados[20] )
   END_RUNG wire#w1
   RUNG wire#powerrail
      Contact( "DB_SUB_1_GENERAL".Estados[22] )
   END_RUNG wire#w1
   RUNG wire#powerrail
      Contact( "DB_SUB_1_GENERAL".Estados[23] )
   END_RUNG wire#w1
   RUNG wire#powerrail
      Contact( "DB_SUB_1_GENERAL".Estados[24] )
   END_RUNG wire#w1
   // the same network as SCL:
   "02_LINEA_Salidas-DB".EnMarcha := ("DB_SUB_1_GENERAL".Estados[1] OR "DB_SUB_1_GENERAL".Estados[2] OR "DB_SUB_1_GENERAL".Estados[3] OR "DB_SUB_1_GENERAL".Estados[4] OR "DB_SUB_1_GENERAL".Estados[5] OR "DB_SUB_1_GENERAL".Estados[6] OR "DB_SUB_1_GENERAL".Estados[7] OR "DB_SUB_1_GENERAL".Estados[8] OR "DB_SUB_1_GENERAL".Estados[9] OR "DB_SUB_1_GENERAL".Estados[10] OR "DB_SUB_1_GENERAL".Estados[11] OR "DB_SUB_1_GENERAL".Estados[12] OR "DB_SUB_1_GENERAL".Estados[13] OR "DB_SUB_1_GENERAL".Estados[14] OR "DB_SUB_1_GENERAL".Estados[15] OR "DB_SUB_1_GENERAL".Estados[16] OR "DB_SUB_1_GENERAL".Estados[17] OR "DB_SUB_1_GENERAL".Estados[18] OR "DB_SUB_1_GENERAL".Estados[19] OR "DB_SUB_1_GENERAL".Estados[20] OR "DB_SUB_1_GENERAL".Estados[22] OR "DB_SUB_1_GENERAL".Estados[23] OR "DB_SUB_1_GENERAL".Estados[24]) AND "01_LINEA_Entradas-DB".Hab_Inverter AND NOT "02_LINEA_Salidas-DB".EnFalla AND "01_LINEA_Entradas-DB".Enc_andando AND NOT "01_LINEA_Entradas-DB".Enc_parada AND NOT "02_LINEA_Salidas-DB".Alarma_Sonora;
END_REGION

REGION Network 64: Testigo de divider en marcha
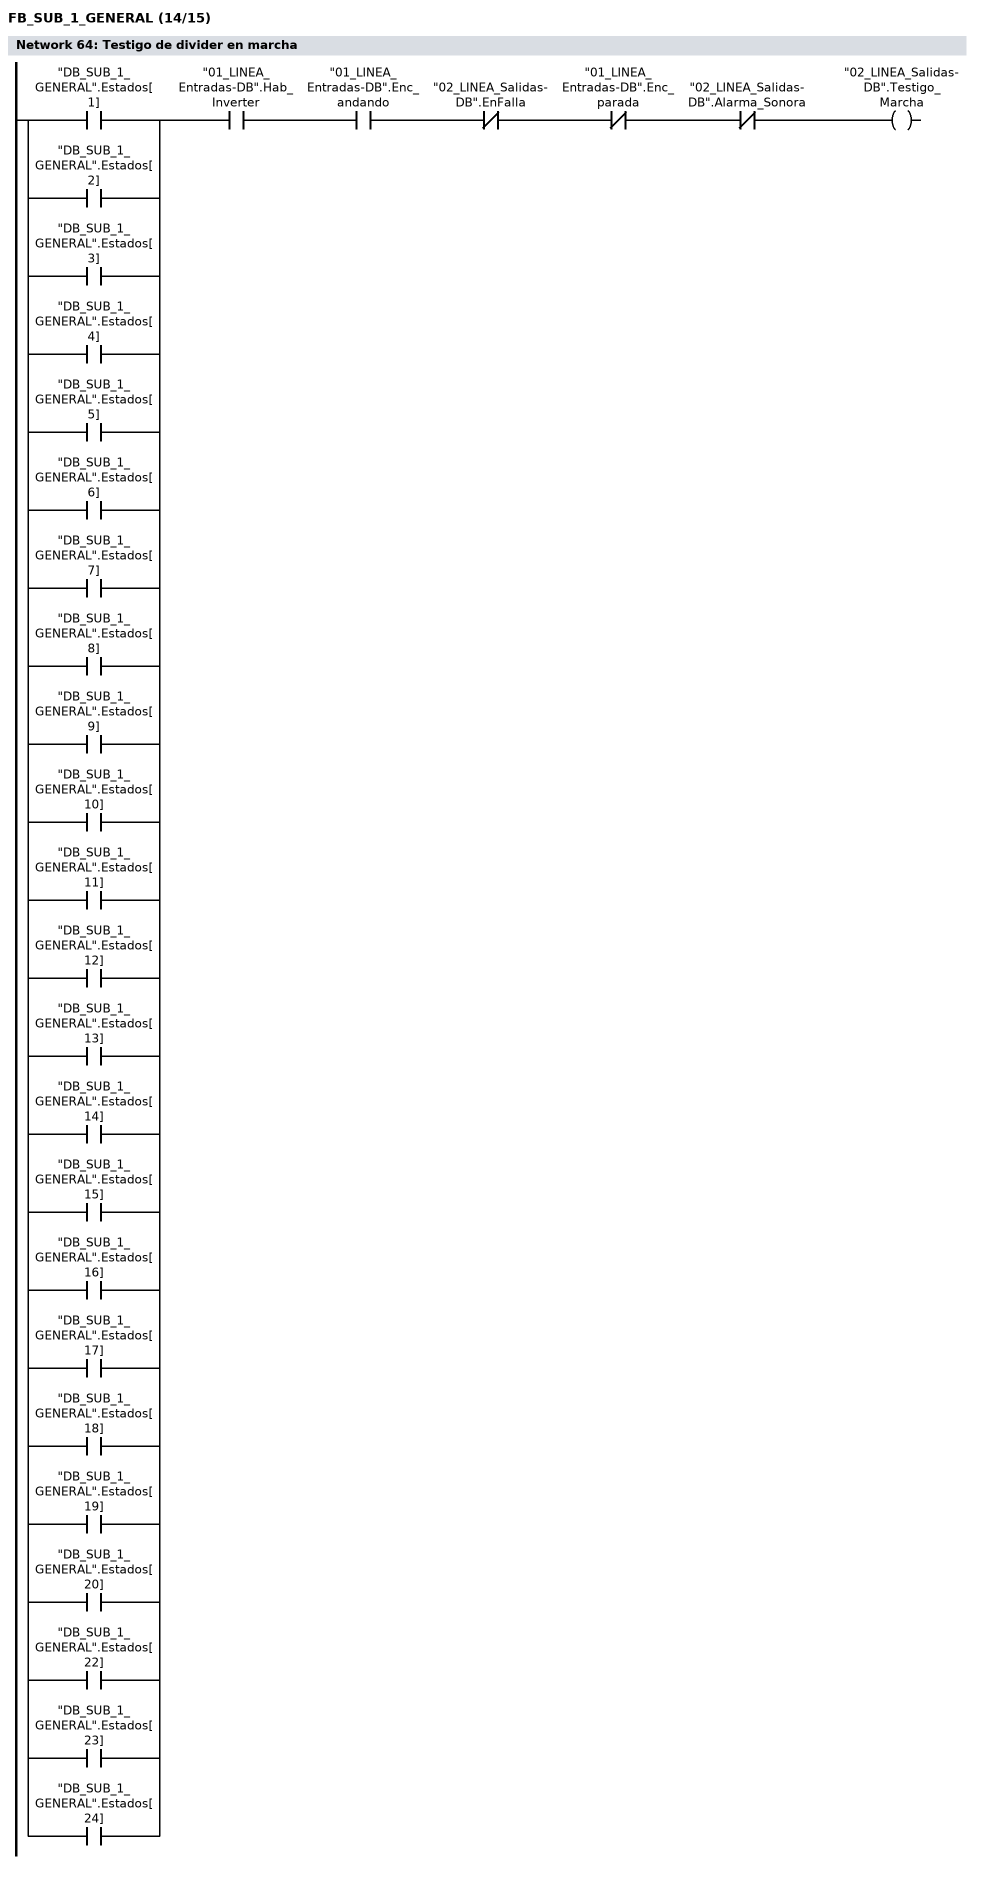
   RUNG wire#powerrail
      Contact( "DB_SUB_1_GENERAL".Estados[1] )
      wire#w1
      Contact( "01_LINEA_Entradas-DB".Hab_Inverter )
      Contact( "01_LINEA_Entradas-DB".Enc_andando )
      I_Contact( "02_LINEA_Salidas-DB".EnFalla )
      I_Contact( "01_LINEA_Entradas-DB".Enc_parada )
      I_Contact( "02_LINEA_Salidas-DB".Alarma_Sonora )
      Coil( "02_LINEA_Salidas-DB".Testigo_Marcha )
   END_RUNG
   RUNG wire#powerrail
      Contact( "DB_SUB_1_GENERAL".Estados[2] )
   END_RUNG wire#w1
   RUNG wire#powerrail
      Contact( "DB_SUB_1_GENERAL".Estados[3] )
   END_RUNG wire#w1
   RUNG wire#powerrail
      Contact( "DB_SUB_1_GENERAL".Estados[4] )
   END_RUNG wire#w1
   RUNG wire#powerrail
      Contact( "DB_SUB_1_GENERAL".Estados[5] )
   END_RUNG wire#w1
   RUNG wire#powerrail
      Contact( "DB_SUB_1_GENERAL".Estados[6] )
   END_RUNG wire#w1
   RUNG wire#powerrail
      Contact( "DB_SUB_1_GENERAL".Estados[7] )
   END_RUNG wire#w1
   RUNG wire#powerrail
      Contact( "DB_SUB_1_GENERAL".Estados[8] )
   END_RUNG wire#w1
   RUNG wire#powerrail
      Contact( "DB_SUB_1_GENERAL".Estados[9] )
   END_RUNG wire#w1
   RUNG wire#powerrail
      Contact( "DB_SUB_1_GENERAL".Estados[10] )
   END_RUNG wire#w1
   RUNG wire#powerrail
      Contact( "DB_SUB_1_GENERAL".Estados[11] )
   END_RUNG wire#w1
   RUNG wire#powerrail
      Contact( "DB_SUB_1_GENERAL".Estados[12] )
   END_RUNG wire#w1
   RUNG wire#powerrail
      Contact( "DB_SUB_1_GENERAL".Estados[13] )
   END_RUNG wire#w1
   RUNG wire#powerrail
      Contact( "DB_SUB_1_GENERAL".Estados[14] )
   END_RUNG wire#w1
   RUNG wire#powerrail
      Contact( "DB_SUB_1_GENERAL".Estados[15] )
   END_RUNG wire#w1
   RUNG wire#powerrail
      Contact( "DB_SUB_1_GENERAL".Estados[16] )
   END_RUNG wire#w1
   RUNG wire#powerrail
      Contact( "DB_SUB_1_GENERAL".Estados[17] )
   END_RUNG wire#w1
   RUNG wire#powerrail
      Contact( "DB_SUB_1_GENERAL".Estados[18] )
   END_RUNG wire#w1
   RUNG wire#powerrail
      Contact( "DB_SUB_1_GENERAL".Estados[19] )
   END_RUNG wire#w1
   RUNG wire#powerrail
      Contact( "DB_SUB_1_GENERAL".Estados[20] )
   END_RUNG wire#w1
   RUNG wire#powerrail
      Contact( "DB_SUB_1_GENERAL".Estados[22] )
   END_RUNG wire#w1
   RUNG wire#powerrail
      Contact( "DB_SUB_1_GENERAL".Estados[23] )
   END_RUNG wire#w1
   RUNG wire#powerrail
      Contact( "DB_SUB_1_GENERAL".Estados[24] )
   END_RUNG wire#w1
   // the same network as SCL:
   "02_LINEA_Salidas-DB".Testigo_Marcha := ("DB_SUB_1_GENERAL".Estados[1] OR "DB_SUB_1_GENERAL".Estados[2] OR "DB_SUB_1_GENERAL".Estados[3] OR "DB_SUB_1_GENERAL".Estados[4] OR "DB_SUB_1_GENERAL".Estados[5] OR "DB_SUB_1_GENERAL".Estados[6] OR "DB_SUB_1_GENERAL".Estados[7] OR "DB_SUB_1_GENERAL".Estados[8] OR "DB_SUB_1_GENERAL".Estados[9] OR "DB_SUB_1_GENERAL".Estados[10] OR "DB_SUB_1_GENERAL".Estados[11] OR "DB_SUB_1_GENERAL".Estados[12] OR "DB_SUB_1_GENERAL".Estados[13] OR "DB_SUB_1_GENERAL".Estados[14] OR "DB_SUB_1_GENERAL".Estados[15] OR "DB_SUB_1_GENERAL".Estados[16] OR "DB_SUB_1_GENERAL".Estados[17] OR "DB_SUB_1_GENERAL".Estados[18] OR "DB_SUB_1_GENERAL".Estados[19] OR "DB_SUB_1_GENERAL".Estados[20] OR "DB_SUB_1_GENERAL".Estados[22] OR "DB_SUB_1_GENERAL".Estados[23] OR "DB_SUB_1_GENERAL".Estados[24]) AND "01_LINEA_Entradas-DB".Hab_Inverter AND "01_LINEA_Entradas-DB".Enc_andando AND NOT "02_LINEA_Salidas-DB".EnFalla AND NOT "01_LINEA_Entradas-DB".Enc_parada AND NOT "02_LINEA_Salidas-DB".Alarma_Sonora;
END_REGION

REGION Network 65: Semaforo verde
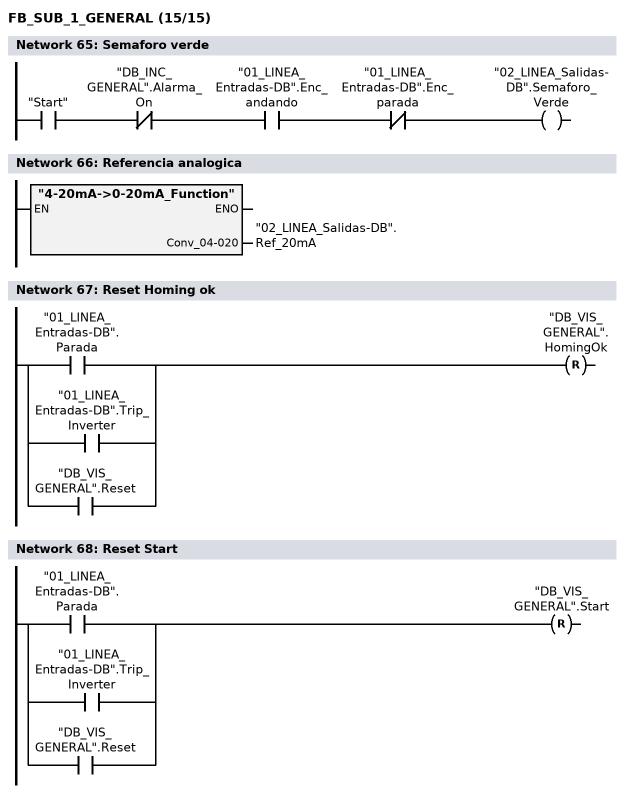
   RUNG wire#powerrail
      Contact( "Start" )
      I_Contact( "DB_INC_GENERAL".Alarma_On )
      Contact( "01_LINEA_Entradas-DB".Enc_andando )
      I_Contact( "01_LINEA_Entradas-DB".Enc_parada )
      Coil( "02_LINEA_Salidas-DB".Semaforo_Verde )
   END_RUNG
   // the same network as SCL:
   "02_LINEA_Salidas-DB".Semaforo_Verde := "Start" AND NOT "DB_INC_GENERAL".Alarma_On AND "01_LINEA_Entradas-DB".Enc_andando AND NOT "01_LINEA_Entradas-DB".Enc_parada;
END_REGION

REGION Network 66: Referencia analogica
   RUNG wire#powerrail
      "4-20mA->0-20mA_Function"("Conv_04-020" => "02_LINEA_Salidas-DB".Ref_20mA)
   END_RUNG
   // the same network as SCL:
   "4-20mA->0-20mA_Function"("Conv_04-020" => "02_LINEA_Salidas-DB".Ref_20mA);
END_REGION

REGION Network 67: Reset Homing ok
   RUNG wire#powerrail
      Contact( "01_LINEA_Entradas-DB".Parada )
      wire#w1
      R_Coil( "DB_VIS_GENERAL".HomingOk )
   END_RUNG
   RUNG wire#powerrail
      Contact( "01_LINEA_Entradas-DB".Trip_Inverter )
   END_RUNG wire#w1
   RUNG wire#powerrail
      Contact( "DB_VIS_GENERAL".Reset )
   END_RUNG wire#w1
   // the same network as SCL:
   IF "01_LINEA_Entradas-DB".Parada OR "01_LINEA_Entradas-DB".Trip_Inverter OR "DB_VIS_GENERAL".Reset THEN
       "DB_VIS_GENERAL".HomingOk := FALSE;
   END_IF;
END_REGION

REGION Network 68: Reset Start
   RUNG wire#powerrail
      Contact( "01_LINEA_Entradas-DB".Parada )
      wire#w1
      R_Coil( "DB_VIS_GENERAL".Start )
   END_RUNG
   RUNG wire#powerrail
      Contact( "01_LINEA_Entradas-DB".Trip_Inverter )
   END_RUNG wire#w1
   RUNG wire#powerrail
      Contact( "DB_VIS_GENERAL".Reset )
   END_RUNG wire#w1
   // the same network as SCL:
   IF "01_LINEA_Entradas-DB".Parada OR "01_LINEA_Entradas-DB".Trip_Inverter OR "DB_VIS_GENERAL".Reset THEN
       "DB_VIS_GENERAL".Start := FALSE;
   END_IF;
END_REGION
END_FUNCTION_BLOCK

FUNCTION "01_LINEA_Entradas" : Void   // FC1, LAD
TITLE = Bloque de entradas
{ S7_Optimized_Access := 'TRUE' }
VERSION : 0.1
BEGIN

REGION Network 1: Contador
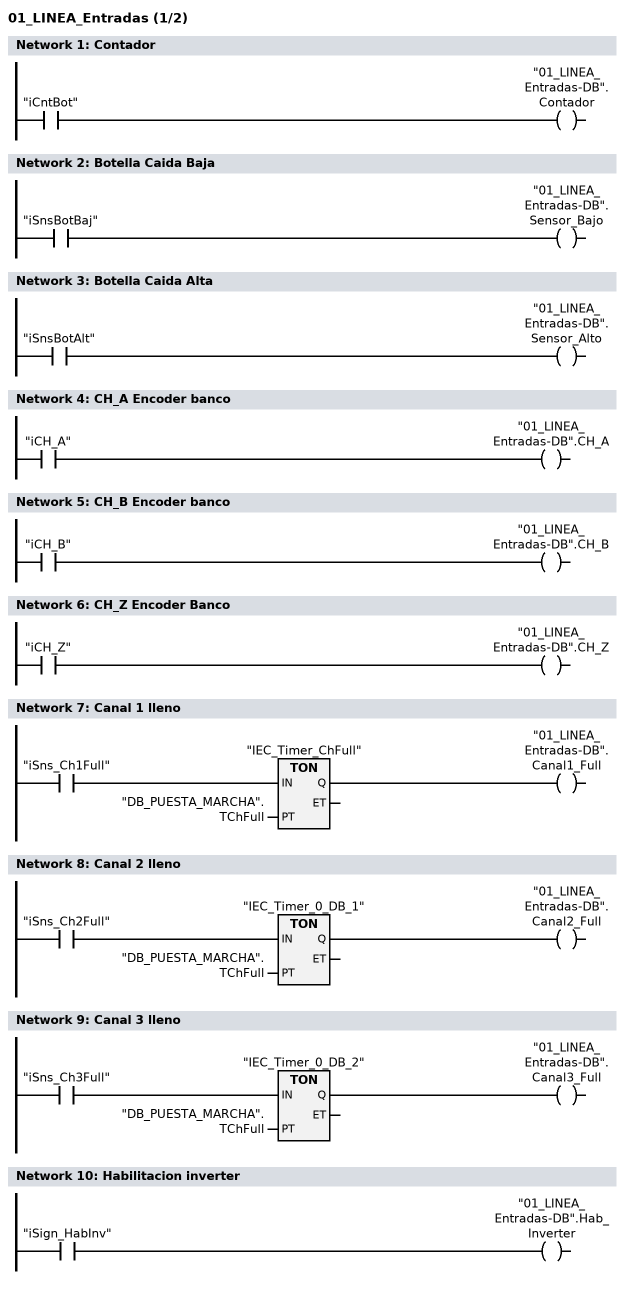
   RUNG wire#powerrail
      Contact( "iCntBot" )
      Coil( "01_LINEA_Entradas-DB".Contador )
   END_RUNG
   // the same network as SCL:
   "01_LINEA_Entradas-DB".Contador := "iCntBot";
END_REGION

REGION Network 2: Botella Caida Baja
   RUNG wire#powerrail
      Contact( "iSnsBotBaj" )
      Coil( "01_LINEA_Entradas-DB".Sensor_Bajo )
   END_RUNG
   // the same network as SCL:
   "01_LINEA_Entradas-DB".Sensor_Bajo := "iSnsBotBaj";
END_REGION

REGION Network 3: Botella Caida Alta
   RUNG wire#powerrail
      Contact( "iSnsBotAlt" )
      Coil( "01_LINEA_Entradas-DB".Sensor_Alto )
   END_RUNG
   // the same network as SCL:
   "01_LINEA_Entradas-DB".Sensor_Alto := "iSnsBotAlt";
END_REGION

REGION Network 4: CH_A Encoder banco
   RUNG wire#powerrail
      Contact( "iCH_A" )
      Coil( "01_LINEA_Entradas-DB".CH_A )
   END_RUNG
   // the same network as SCL:
   "01_LINEA_Entradas-DB".CH_A := "iCH_A";
END_REGION

REGION Network 5: CH_B Encoder banco
   RUNG wire#powerrail
      Contact( "iCH_B" )
      Coil( "01_LINEA_Entradas-DB".CH_B )
   END_RUNG
   // the same network as SCL:
   "01_LINEA_Entradas-DB".CH_B := "iCH_B";
END_REGION

REGION Network 6: CH_Z Encoder Banco
   RUNG wire#powerrail
      Contact( "iCH_Z" )
      Coil( "01_LINEA_Entradas-DB".CH_Z )
   END_RUNG
   // the same network as SCL:
   "01_LINEA_Entradas-DB".CH_Z := "iCH_Z";
END_REGION

REGION Network 7: Canal 1 lleno
   "IEC_Timer_ChFull".TON(IN := "iSns_Ch1Full", PT := "DB_PUESTA_MARCHA".TChFull);
   "01_LINEA_Entradas-DB".Canal1_Full := "IEC_Timer_ChFull".Q;
END_REGION

REGION Network 8: Canal 2 lleno
   "IEC_Timer_0_DB_1".TON(IN := "iSns_Ch2Full", PT := "DB_PUESTA_MARCHA".TChFull);
   "01_LINEA_Entradas-DB".Canal2_Full := "IEC_Timer_0_DB_1".Q;
END_REGION

REGION Network 9: Canal 3 lleno
   "IEC_Timer_0_DB_2".TON(IN := "iSns_Ch3Full", PT := "DB_PUESTA_MARCHA".TChFull);
   "01_LINEA_Entradas-DB".Canal3_Full := "IEC_Timer_0_DB_2".Q;
END_REGION

REGION Network 10: Habilitacion inverter
   RUNG wire#powerrail
      Contact( "iSign_HabInv" )
      Coil( "01_LINEA_Entradas-DB".Hab_Inverter )
   END_RUNG
   // the same network as SCL:
   "01_LINEA_Entradas-DB".Hab_Inverter := "iSign_HabInv";
END_REGION

REGION Network 11: Pulsador de Marcha de la columna 11
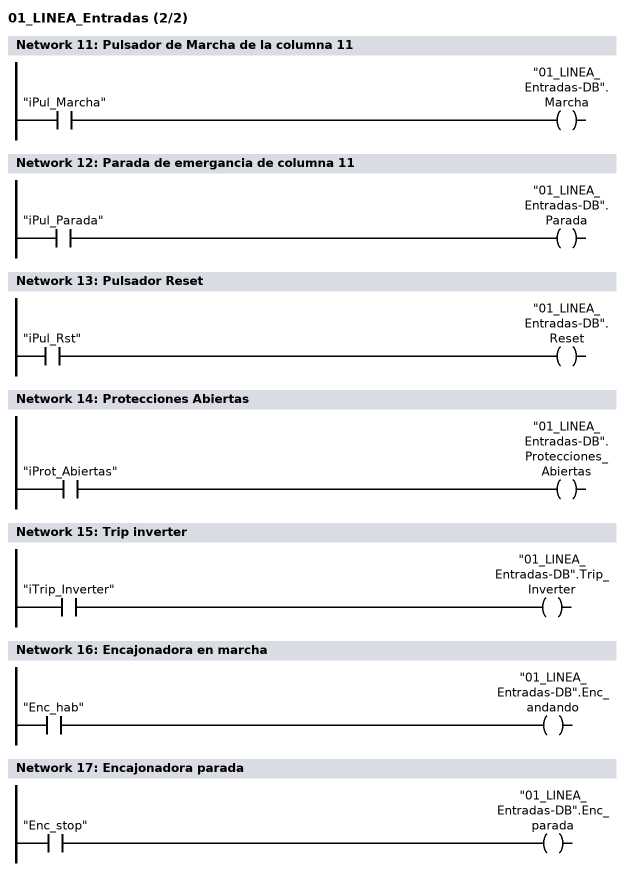
   RUNG wire#powerrail
      Contact( "iPul_Marcha" )
      Coil( "01_LINEA_Entradas-DB".Marcha )
   END_RUNG
   // the same network as SCL:
   "01_LINEA_Entradas-DB".Marcha := "iPul_Marcha";
END_REGION

REGION Network 12: Parada de emergancia de columna 11
   RUNG wire#powerrail
      Contact( "iPul_Parada" )
      Coil( "01_LINEA_Entradas-DB".Parada )
   END_RUNG
   // the same network as SCL:
   "01_LINEA_Entradas-DB".Parada := "iPul_Parada";
END_REGION

REGION Network 13: Pulsador Reset
   RUNG wire#powerrail
      Contact( "iPul_Rst" )
      Coil( "01_LINEA_Entradas-DB".Reset )
   END_RUNG
   // the same network as SCL:
   "01_LINEA_Entradas-DB".Reset := "iPul_Rst";
END_REGION

REGION Network 14: Protecciones Abiertas
   RUNG wire#powerrail
      Contact( "iProt_Abiertas" )
      Coil( "01_LINEA_Entradas-DB".Protecciones_Abiertas )
   END_RUNG
   // the same network as SCL:
   "01_LINEA_Entradas-DB".Protecciones_Abiertas := "iProt_Abiertas";
END_REGION

REGION Network 15: Trip inverter
   RUNG wire#powerrail
      Contact( "iTrip_Inverter" )
      Coil( "01_LINEA_Entradas-DB".Trip_Inverter )
   END_RUNG
   // the same network as SCL:
   "01_LINEA_Entradas-DB".Trip_Inverter := "iTrip_Inverter";
END_REGION

REGION Network 16: Encajonadora en marcha
   RUNG wire#powerrail
      Contact( "Enc_hab" )
      Coil( "01_LINEA_Entradas-DB".Enc_andando )
   END_RUNG
   // the same network as SCL:
   "01_LINEA_Entradas-DB".Enc_andando := "Enc_hab";
END_REGION

REGION Network 17: Encajonadora parada
   RUNG wire#powerrail
      Contact( "Enc_stop" )
      Coil( "01_LINEA_Entradas-DB".Enc_parada )
   END_RUNG
   // the same network as SCL:
   "01_LINEA_Entradas-DB".Enc_parada := "Enc_stop";
END_REGION
END_FUNCTION

FUNCTION "02_LINEA_Salidas" : Void   // FC2, LAD
{ S7_Optimized_Access := 'TRUE' }
VERSION : 0.1
BEGIN

REGION Network 1: Alarma Sonora
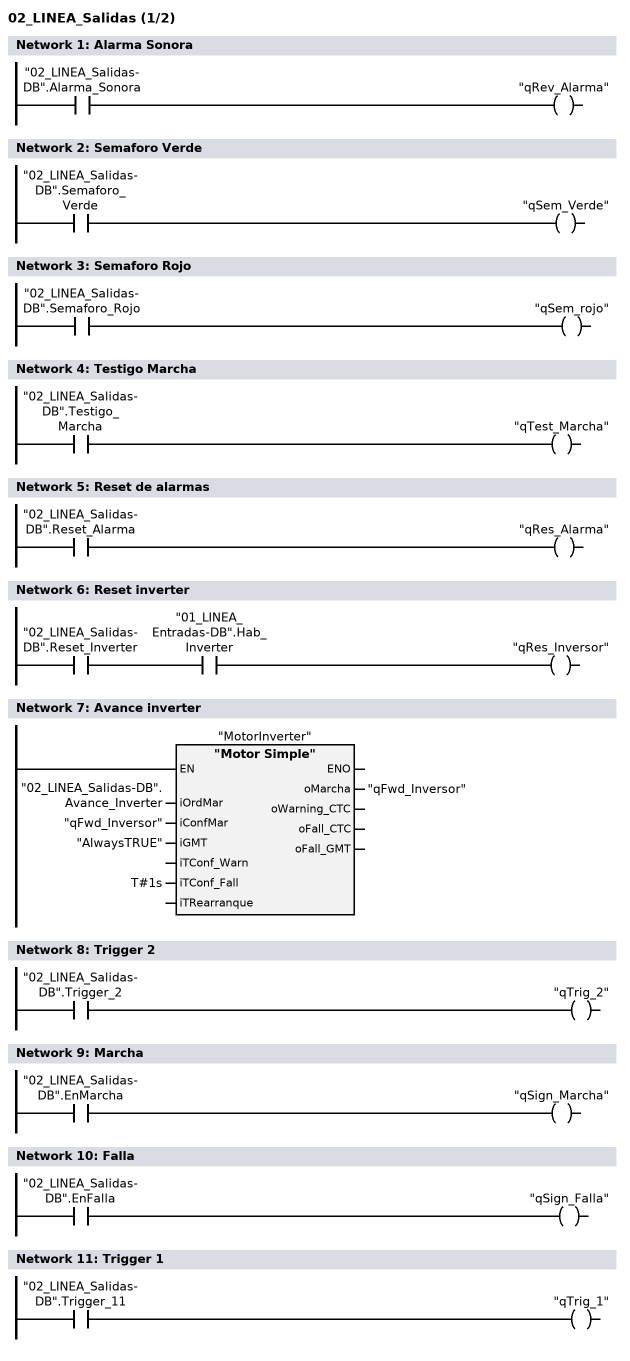
   RUNG wire#powerrail
      Contact( "02_LINEA_Salidas-DB".Alarma_Sonora )
      Coil( "qRev_Alarma" )
   END_RUNG
   // the same network as SCL:
   "qRev_Alarma" := "02_LINEA_Salidas-DB".Alarma_Sonora;
END_REGION

REGION Network 2: Semaforo Verde
   RUNG wire#powerrail
      Contact( "02_LINEA_Salidas-DB".Semaforo_Verde )
      Coil( "qSem_Verde" )
   END_RUNG
   // the same network as SCL:
   "qSem_Verde" := "02_LINEA_Salidas-DB".Semaforo_Verde;
END_REGION

REGION Network 3: Semaforo Rojo
   RUNG wire#powerrail
      Contact( "02_LINEA_Salidas-DB".Semaforo_Rojo )
      Coil( "qSem_rojo" )
   END_RUNG
   // the same network as SCL:
   "qSem_rojo" := "02_LINEA_Salidas-DB".Semaforo_Rojo;
END_REGION

REGION Network 4: Testigo Marcha
   RUNG wire#powerrail
      Contact( "02_LINEA_Salidas-DB".Testigo_Marcha )
      Coil( "qTest_Marcha" )
   END_RUNG
   // the same network as SCL:
   "qTest_Marcha" := "02_LINEA_Salidas-DB".Testigo_Marcha;
END_REGION

REGION Network 5: Reset de alarmas
   RUNG wire#powerrail
      Contact( "02_LINEA_Salidas-DB".Reset_Alarma )
      Coil( "qRes_Alarma" )
   END_RUNG
   // the same network as SCL:
   "qRes_Alarma" := "02_LINEA_Salidas-DB".Reset_Alarma;
END_REGION

REGION Network 6: Reset inverter
   RUNG wire#powerrail
      Contact( "02_LINEA_Salidas-DB".Reset_Inverter )
      Contact( "01_LINEA_Entradas-DB".Hab_Inverter )
      Coil( "qRes_Inversor" )
   END_RUNG
   // the same network as SCL:
   "qRes_Inversor" := "02_LINEA_Salidas-DB".Reset_Inverter AND "01_LINEA_Entradas-DB".Hab_Inverter;
END_REGION

REGION Network 7: Avance inverter
   RUNG wire#powerrail
      "MotorInverter"(iOrdMar := "02_LINEA_Salidas-DB".Avance_Inverter, iConfMar := "qFwd_Inversor", iGMT := "AlwaysTRUE", iTConf_Warn :=, iTConf_Fall := T#1s, iTRearranque :=, oMarcha => "qFwd_Inversor", oWarning_CTC =>, oFall_CTC =>, oFall_GMT =>)
   END_RUNG
   // the same network as SCL:
   "MotorInverter"(iOrdMar := "02_LINEA_Salidas-DB".Avance_Inverter,   // "Motor Simple"
                   iConfMar := "qFwd_Inversor",
                   iGMT := "AlwaysTRUE",
                   iTConf_Fall := T#1s,
                   oMarcha => "qFwd_Inversor");
END_REGION

REGION Network 8: Trigger 2
   RUNG wire#powerrail
      Contact( "02_LINEA_Salidas-DB".Trigger_2 )
      Coil( "qTrig_2" )
   END_RUNG
   // the same network as SCL:
   "qTrig_2" := "02_LINEA_Salidas-DB".Trigger_2;
END_REGION

REGION Network 9: Marcha
   RUNG wire#powerrail
      Contact( "02_LINEA_Salidas-DB".EnMarcha )
      Coil( "qSign_Marcha" )
   END_RUNG
   // the same network as SCL:
   "qSign_Marcha" := "02_LINEA_Salidas-DB".EnMarcha;
END_REGION

REGION Network 10: Falla
   RUNG wire#powerrail
      Contact( "02_LINEA_Salidas-DB".EnFalla )
      Coil( "qSign_Falla" )
   END_RUNG
   // the same network as SCL:
   "qSign_Falla" := "02_LINEA_Salidas-DB".EnFalla;
END_REGION

REGION Network 11: Trigger 1
   RUNG wire#powerrail
      Contact( "02_LINEA_Salidas-DB".Trigger_11 )
      Coil( "qTrig_1" )
   END_RUNG
   // the same network as SCL:
   "qTrig_1" := "02_LINEA_Salidas-DB".Trigger_11;
END_REGION

REGION Network 12: Trigger 22
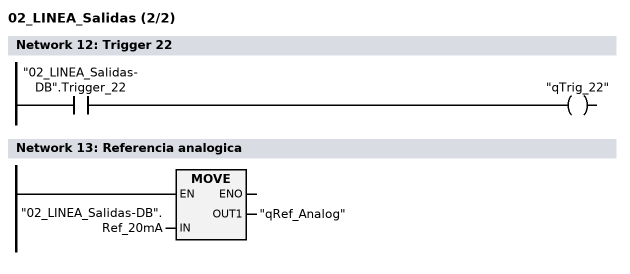
   RUNG wire#powerrail
      Contact( "02_LINEA_Salidas-DB".Trigger_22 )
      Coil( "qTrig_22" )
   END_RUNG
   // the same network as SCL:
   "qTrig_22" := "02_LINEA_Salidas-DB".Trigger_22;
END_REGION

REGION Network 13: Referencia analogica
   RUNG wire#powerrail
      Move(in := "02_LINEA_Salidas-DB".Ref_20mA, out1 => "qRef_Analog")
   END_RUNG
   // the same network as SCL:
   "qRef_Analog" := "02_LINEA_Salidas-DB".Ref_20mA;
END_REGION
END_FUNCTION

FUNCTION "4-20mA->0-20mA_Function" : Void   // FC3, LAD
TITLE = Conversion 4-20 -> 0-20 Canal 1
{ S7_Optimized_Access := 'TRUE' }
VERSION : 0.1
   VAR_OUTPUT
      "Conv_04-020" : Int;
   END_VAR
   VAR_TEMP
      Input_Analog1 : Real;
      Temp_Analog1 : Real;
      Input_Analog2 : Real;
      Temp_Analog2 : Real;
   END_VAR
BEGIN

REGION Network 1
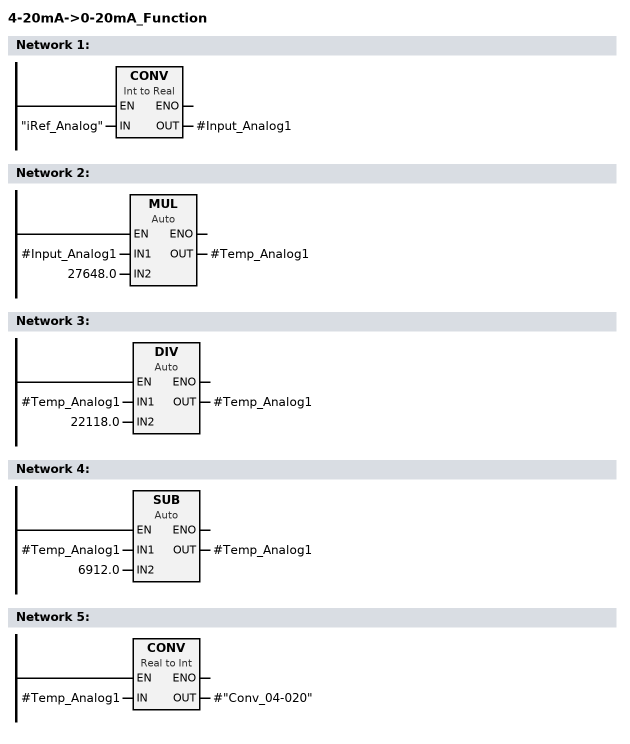
   RUNG wire#powerrail
      { S7_Templates := "[SrcType := Int, DestType := Real]" } Convert(in := "iRef_Analog", out => #Input_Analog1)
   END_RUNG
   // the same network as SCL:
   #Input_Analog1 := INT_TO_REAL("iRef_Analog");
END_REGION

REGION Network 2
   RUNG wire#powerrail
      Mul(in1 := #Input_Analog1, in2 := 27648.0, out => #Temp_Analog1)
   END_RUNG
   // the same network as SCL:
   #Temp_Analog1 := #Input_Analog1 * 27648.0;
END_REGION

REGION Network 3
   RUNG wire#powerrail
      Div(in1 := #Temp_Analog1, in2 := 22118.0, out => #Temp_Analog1)
   END_RUNG
   // the same network as SCL:
   #Temp_Analog1 := #Temp_Analog1 / 22118.0;
END_REGION

REGION Network 4
   RUNG wire#powerrail
      Sub(in1 := #Temp_Analog1, in2 := 6912.0, out => #Temp_Analog1)
   END_RUNG
   // the same network as SCL:
   #Temp_Analog1 := #Temp_Analog1 - 6912.0;
END_REGION

REGION Network 5
   RUNG wire#powerrail
      { S7_Templates := "[SrcType := Real, DestType := Int]" } Convert(in := #Temp_Analog1, out => #"Conv_04-020")
   END_RUNG
   // the same network as SCL:
   #"Conv_04-020" := REAL_TO_INT(#Temp_Analog1);
END_REGION
END_FUNCTION

ORGANIZATION_BLOCK "Main"   // OB1, LAD, ProgramCycle
TITLE = "Main Program Sweep (Cycle)"
{ S7_Optimized_Access := 'TRUE' }
VERSION : 0.1
   VAR_INPUT
      Initial_Call : Bool;   // Initial call of this OB
      Remanence : Bool;   // =True, if remanent data are available
   END_VAR
BEGIN

REGION Network 1: Asigno entradas a variables
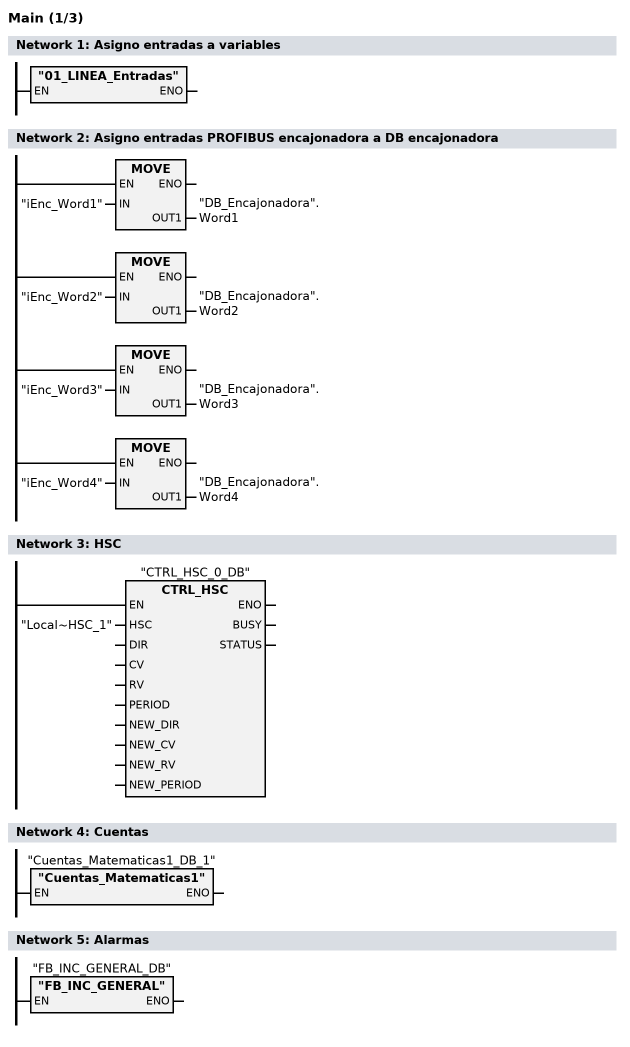
   RUNG wire#powerrail
      "01_LINEA_Entradas"()
   END_RUNG
   // the same network as SCL:
   "01_LINEA_Entradas"();
END_REGION

REGION Network 2: Asigno entradas PROFIBUS encajonadora a DB encajonadora
   RUNG wire#powerrail
      Move(in := "iEnc_Word1", out1 => "DB_Encajonadora".Word1)
   END_RUNG
   RUNG wire#powerrail
      Move(in := "iEnc_Word2", out1 => "DB_Encajonadora".Word2)
   END_RUNG
   RUNG wire#powerrail
      Move(in := "iEnc_Word3", out1 => "DB_Encajonadora".Word3)
   END_RUNG
   RUNG wire#powerrail
      Move(in := "iEnc_Word4", out1 => "DB_Encajonadora".Word4)
   END_RUNG
   // the same network as SCL:
   "DB_Encajonadora".Word1 := "iEnc_Word1";
   "DB_Encajonadora".Word2 := "iEnc_Word2";
   "DB_Encajonadora".Word3 := "iEnc_Word3";
   "DB_Encajonadora".Word4 := "iEnc_Word4";
END_REGION

REGION Network 3: HSC
   "CTRL_HSC_0_DB"(HSC := "Local~HSC_1");   // CTRL_HSC
END_REGION

REGION Network 4: Cuentas
   RUNG wire#powerrail
      "Cuentas_Matematicas1_DB_1"()
   END_RUNG
   // the same network as SCL:
   "Cuentas_Matematicas1_DB_1"();   // "Cuentas_Matematicas1"
END_REGION

REGION Network 5: Alarmas
   RUNG wire#powerrail
      "FB_INC_GENERAL_DB"()
   END_RUNG
   // the same network as SCL:
   "FB_INC_GENERAL_DB"();   // "FB_INC_GENERAL"
END_REGION

REGION Network 6: Habilito ejes
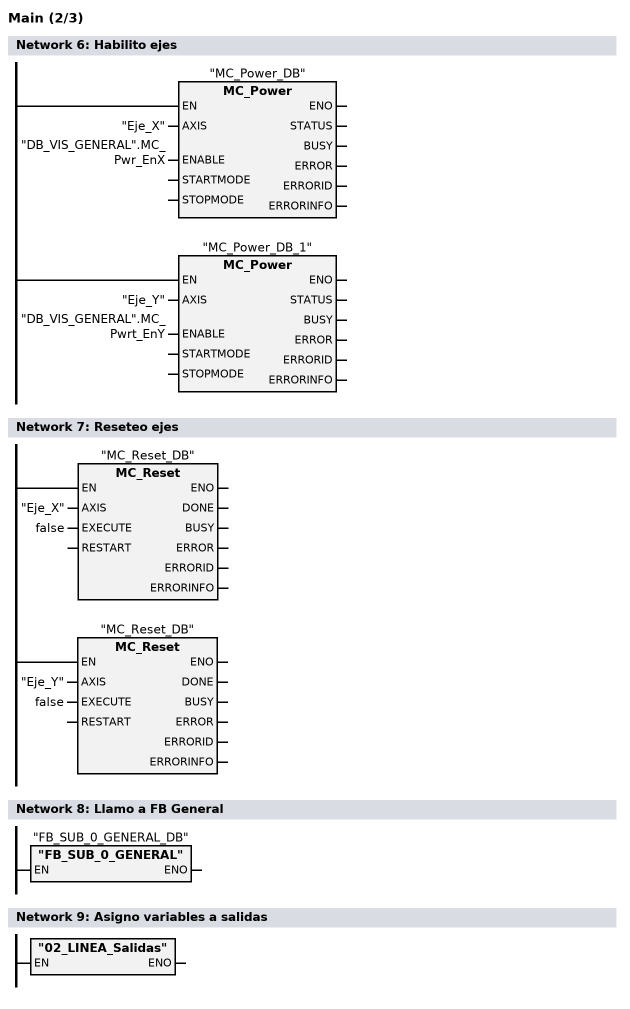
   "MC_Power_DB"(Axis := "Eje_X", Enable := "DB_VIS_GENERAL".MC_Pwr_EnX);   // MC_Power
   "MC_Power_DB_1"(Axis := "Eje_Y", Enable := "DB_VIS_GENERAL".MC_Pwrt_EnY);   // MC_Power
END_REGION

REGION Network 7: Reseteo ejes
   "MC_Reset_DB"(Axis := "Eje_X", Execute := false);   // MC_Reset
   "MC_Reset_DB"(Axis := "Eje_Y", Execute := false);   // MC_Reset
END_REGION

REGION Network 8: Llamo a FB General
   RUNG wire#powerrail
      "FB_SUB_0_GENERAL_DB"()
   END_RUNG
   // the same network as SCL:
   "FB_SUB_0_GENERAL_DB"();   // "FB_SUB_0_GENERAL"
END_REGION

REGION Network 9: Asigno variables a salidas
   RUNG wire#powerrail
      "02_LINEA_Salidas"()
   END_RUNG
   // the same network as SCL:
   "02_LINEA_Salidas"();
END_REGION

REGION Network 10: Asigno DB encajonadora a salidas PROFIBUS
